LIN {X 0,Y 418.249,Z 282.699,A -85,B 0,C 180,E1 -10100.662,E2 -10100.662} C_VEL
LIN {X 0,Y 418.288,Z 282.694,A -85,B 0,C 180,E1 -10103.781,E2 -10103.781} C_VEL
LIN {X 0,Y 418.309,Z 282.695,A -85,B 0,C 180,E1 -10107.07,E2 -10107.07} C_VEL
LIN {X 0,Y 418.243,Z 282.698,A -85,B 0,C 180,E1 -10110.272,E2 -10110.272} C_VEL
LIN {X 0,Y 418.247,Z 282.697,A -85,B 0,C 180,E1 -10113.677,E2 -10113.677} C_VEL
LIN {X 0,Y 418.244,Z 282.692,A -85,B 0,C 180,E1 -10117.223,E2 -10117.223} C_VEL
LIN {X 0,Y 418.251,Z 282.695,A -85,B 0,C 180,E1 -10119.681,E2 -10119.681} C_VEL
LIN {X 0,Y 418.231,Z 282.701,A -85,B 0,C 180,E1 -10122.321,E2 -10122.321} C_VEL
LIN {X 0,Y 418.24,Z 282.698,A -85,B 0,C 180,E1 -10125.109,E2 -10125.109} C_VEL
LIN {X 0,Y 418.24,Z 282.695,A -85,B 0,C 180,E1 -10127.767,E2 -10127.767} C_VEL
LIN {X 0,Y 418.256,Z 282.699,A -85,B 0,C 180,E1 -10130.618,E2 -10130.618} C_VEL
LIN {X 0,Y 418.25,Z 282.714,A -85,B 0,C 180,E1 -10133.881,E2 -10133.881} C_VEL
LIN {X 0,Y 423.641,Z 299.97,A -85,B 0,C 180,E1 -10136.508,E2 -10136.508} C_VEL
LIN {X 0,Y 426.193,Z 308.268,A -85,B 0,C 180,E1 -10137.685,E2 -10137.685} C_VEL
LIN {X 0,Y 432.078,Z 321.178,A -85,B 0,C 180,E1 -10138.364,E2 -10138.364} C_VEL
LIN {X 0,Y 435.625,Z 342.848,A -85,B 0,C 180,E1 -10139.021,E2 -10139.021} C_VEL
LIN {X 0,Y 432.249,Z 513.22,A -85,B 0,C 180,E1 -10141.933,E2 -10141.933} C_VEL
LIN {X 0,Y 431.437,Z 530.001,A -85,B 0,C 180,E1 -10142.371,E2 -10142.371} C_VEL
LIN {X 0,Y 430.361,Z 546.409,A -85,B 0,C 180,E1 -10142.987,E2 -10142.987} C_VEL
LIN {X 0,Y 429.185,Z 561.958,A -85,B 0,C 180,E1 -10143.76,E2 -10143.76} C_VEL
LIN {X 0,Y 427.765,Z 577.137,A -85,B 0,C 180,E1 -10144.712,E2 -10144.712} C_VEL
LIN {X 0,Y 426.267,Z 591.185,A -85,B 0,C 180,E1 -10145.788,E2 -10145.788} C_VEL
LIN {X 0,Y 424.709,Z 605.609,A -85,B 0,C 180,E1 -10147.116,E2 -10147.116} C_VEL
LIN {X 0,Y 423.361,Z 617.281,A -85,B 0,C 180,E1 -10148.376,E2 -10148.376} C_VEL
LIN {X 0,Y 421.85,Z 630.208,A -85,B 0,C 180,E1 -10150.03,E2 -10150.03} C_VEL
LIN {X 0,Y 420.534,Z 641.484,A -85,B 0,C 180,E1 -10151.739,E2 -10151.739} C_VEL
LIN {X 0,Y 419.547,Z 651.141,A -85,B 0,C 180,E1 -10153.455,E2 -10153.455} C_VEL
LIN {X 0,Y 418.597,Z 660.507,A -85,B 0,C 180,E1 -10155.414,E2 -10155.414} C_VEL
LIN {X 0,Y 417.976,Z 668.29,A -85,B 0,C 180,E1 -10157.374,E2 -10157.374} C_VEL
LIN {X 0,Y 417.475,Z 674.7,A -85,B 0,C 180,E1 -10159.328,E2 -10159.328} C_VEL
LIN {X 0,Y 417.212,Z 679.955,A -85,B 0,C 180,E1 -10161.28,E2 -10161.28} C_VEL
LIN {X 0,Y 417.137,Z 684.944,A -85,B 0,C 180,E1 -10163.739,E2 -10163.739} C_VEL
LIN {X 0,Y 416.984,Z 688.178,A -85,B 0,C 180,E1 -10166.134,E2 -10166.134} C_VEL
LIN {X 0,Y 417.046,Z 689.646,A -85,B 0,C 180,E1 -10168.069,E2 -10168.069} C_VEL
LIN {X 0,Y 416.999,Z 690.206,A -85,B 0,C 180,E1 -10170,E2 -10170} C_VEL
LIN {X 0,Y 417.059,Z 689.728,A -85,B 0,C 180,E1 -10171.932,E2 -10171.932} C_VEL
LIN {X 0,Y 416.982,Z 688.348,A -85,B 0,C 180,E1 -10173.866,E2 -10173.866} C_VEL
LIN {X 0,Y 417.137,Z 685.222,A -85,B 0,C 180,E1 -10176.261,E2 -10176.261} C_VEL
LIN {X 0,Y 417.183,Z 681.492,A -85,B 0,C 180,E1 -10178.233,E2 -10178.233} C_VEL
LIN {X 0,Y 417.397,Z 676.77,A -85,B 0,C 180,E1 -10180.183,E2 -10180.183} C_VEL
LIN {X 0,Y 417.89,Z 670.825,A -85,B 0,C 180,E1 -10182.136,E2 -10182.136} C_VEL
LIN {X 0,Y 418.552,Z 662.671,A -85,B 0,C 180,E1 -10184.34,E2 -10184.34} C_VEL
LIN {X 0,Y 419.584,Z 653.944,A -85,B 0,C 180,E1 -10186.294,E2 -10186.294} C_VEL
LIN {X 0,Y 420.748,Z 643.558,A -85,B 0,C 180,E1 -10188.252,E2 -10188.252} C_VEL
LIN {X 0,Y 422.177,Z 632.774,A -85,B 0,C 180,E1 -10189.954,E2 -10189.954} C_VEL
LIN {X 0,Y 423.752,Z 620.449,A -85,B 0,C 180,E1 -10191.617,E2 -10191.617} C_VEL
LIN {X 0,Y 425.414,Z 607.474,A -85,B 0,C 180,E1 -10193.102,E2 -10193.102} C_VEL
LIN {X 0,Y 427.132,Z 593.835,A -85,B 0,C 180,E1 -10194.419,E2 -10194.419} C_VEL
LIN {X 0,Y 428.934,Z 578.449,A -85,B 0,C 180,E1 -10195.645,E2 -10195.645} C_VEL
LIN {X 0,Y 430.648,Z 562.514,A -85,B 0,C 180,E1 -10196.666,E2 -10196.666} C_VEL
LIN {X 0,Y 431.982,Z 547.62,A -85,B 0,C 180,E1 -10197.427,E2 -10197.427} C_VEL
LIN {X 0,Y 433.199,Z 531.35,A -85,B 0,C 180,E1 -10198.066,E2 -10198.066} C_VEL
LIN {X 0,Y 434.124,Z 514.455,A -85,B 0,C 180,E1 -10198.532,E2 -10198.532} C_VEL
LIN {X 0,Y 438.122,Z 343.991,A -85,B 0,C 180,E1 -10201.515,E2 -10201.515} C_VEL
LIN {X 0,Y 437.367,Z 337.587,A -85,B 0,C 180,E1 -10201.708,E2 -10201.708} C_VEL
LIN {X 0,Y 434.883,Z 323.612,A -85,B 0,C 180,E1 -10202.21,E2 -10202.21} C_VEL
LIN {X 0,Y 426.694,Z 307.126,A -85,B 0,C 180,E1 -10203.348,E2 -10203.348} C_VEL
LIN {X 0,Y 422.578,Z 294.815,A -85,B 0,C 180,E1 -10205.42,E2 -10205.42} C_VEL
LIN {X 0,Y 418.253,Z 282.699,A -85,B 0,C 180,E1 -10207.639,E2 -10207.639} C_VEL
LIN {X 0,Y 418.223,Z 282.701,A -85,B 0,C 180,E1 -10210.948,E2 -10210.948} C_VEL
LIN {X 0,Y 418.216,Z 282.702,A -85,B 0,C 180,E1 -10213.731,E2 -10213.731} C_VEL
LIN {X 0,Y 418.208,Z 282.702,A -85,B 0,C 180,E1 -10216.449,E2 -10216.449} C_VEL
LIN {X 0,Y 418.223,Z 282.692,A -85,B 0,C 180,E1 -10219.131,E2 -10219.131} C_VEL
LIN {X 0,Y 418.228,Z 282.69,A -85,B 0,C 180,E1 -10222.167,E2 -10222.167} C_VEL
LIN {X 0,Y 418.265,Z 282.693,A -85,B 0,C 180,E1 -10225.42,E2 -10225.42} C_VEL
LIN {X 0,Y 418.211,Z 282.699,A -85,B 0,C 180,E1 -10228.604,E2 -10228.604} C_VEL
LIN {X 0,Y 418.292,Z 282.672,A -85,B 0,C 180,E1 -10231.937,E2 -10231.937} C_VEL
LIN {X 0,Y 418.29,Z 282.69,A -85,B 0,C 180,E1 -10235.163,E2 -10235.163} C_VEL
LIN {X 0,Y 418.235,Z 282.685,A -85,B 0,C 180,E1 -10238.304,E2 -10238.304} C_VEL
LIN {X 0,Y 418.284,Z 282.687,A -85,B 0,C 180,E1 -10241.384,E2 -10241.384} C_VEL
LIN {X 0,Y 418.303,Z 282.677,A -85,B 0,C 180,E1 -10244.406,E2 -10244.406} C_VEL
LIN {X 0,Y 418.357,Z 282.679,A -85,B 0,C 180,E1 -10247.386,E2 -10247.386} C_VEL
LIN {X 0,Y 418.339,Z 282.668,A -85,B 0,C 180,E1 -10250.329,E2 -10250.329} C_VEL
LIN {X 0,Y 418.446,Z 282.67,A -85,B 0,C 180,E1 -10253.249,E2 -10253.249} C_VEL
LIN {X 0,Y 418.331,Z 282.664,A -85,B 0,C 180,E1 -10255.182,E2 -10255.182} C_VEL
LIN {X 0,Y 418.542,Z 282.658,A -85,B 0,C 180,E1 -10258.076,E2 -10258.076} C_VEL
LIN {X 0,Y 418.666,Z 282.644,A -85,B 0,C 180,E1 -10260.001,E2 -10260.001} C_VEL
LIN {X 0,Y 418.475,Z 282.654,A -85,B 0,C 180,E1 -10262.888,E2 -10262.888} C_VEL
LIN {X 0,Y 418.445,Z 282.663,A -85,B 0,C 180,E1 -10266.551,E2 -10266.551} C_VEL
LIN {X 0,Y 418.337,Z 282.679,A -85,B 0,C 180,E1 -10269.672,E2 -10269.672} C_VEL
LIN {X 0,Y 418.349,Z 282.671,A -85,B 0,C 180,E1 -10273.001,E2 -10273.001} C_VEL
LIN {X 0,Y 418.267,Z 282.696,A -85,B 0,C 180,E1 -10276.713,E2 -10276.713} C_VEL
LIN {X 0,Y 418.273,Z 282.679,A -85,B 0,C 180,E1 -10279.79,E2 -10279.79} C_VEL
LIN {X 0,Y 418.227,Z 282.694,A -85,B 0,C 180,E1 -10282.737,E2 -10282.737} C_VEL
LIN {X 0,Y 418.212,Z 282.703,A -85,B 0,C 180,E1 -10285.909,E2 -10285.909} C_VEL
LIN {X 0,Y 418.257,Z 282.692,A -85,B 0,C 180,E1 -10289.163,E2 -10289.163} C_VEL
LIN {X 0,Y 418.233,Z 282.693,A -85,B 0,C 180,E1 -10292.53,E2 -10292.53} C_VEL
LIN {X 0,Y 418.249,Z 282.695,A -85,B 0,C 180,E1 -10294.843,E2 -10294.843} C_VEL
LIN {X 0,Y 418.234,Z 282.695,A -85,B 0,C 180,E1 -10298.445,E2 -10298.445} C_VEL
LIN {X 0,Y 418.249,Z 282.867,A -85,B 0,C 180,E1 -10302.071,E2 -10302.071} C_VEL
LIN {X 0,Y 420.134,Z 288.122,A -85,B 0,C 180,E1 -10303.057,E2 -10303.057} C_VEL
LIN {X 0,Y 429.975,Z 305.451,A -85,B 0,C 180,E1 -10304.41,E2 -10304.41} C_VEL
LIN {X 0,Y 438.474,Z 322.374,A -85,B 0,C 180,E1 -10305.542,E2 -10305.542} C_VEL
LIN {X 0,Y 434.474,Z 493.566,A -85,B 0,C 180,E1 -10308.551,E2 -10308.551} C_VEL
LIN {X 0,Y 433.607,Z 510.226,A -85,B 0,C 180,E1 -10309.029,E2 -10309.029} C_VEL
LIN {X 0,Y 432.602,Z 524.979,A -85,B 0,C 180,E1 -10309.62,E2 -10309.62} C_VEL
LIN {X 0,Y 431.281,Z 540.752,A -85,B 0,C 180,E1 -10310.438,E2 -10310.438} C_VEL
LIN {X 0,Y 429.944,Z 554.135,A -85,B 0,C 180,E1 -10311.3,E2 -10311.3} C_VEL
LIN {X 0,Y 428.353,Z 568.136,A -85,B 0,C 180,E1 -10312.39,E2 -10312.39} C_VEL
LIN {X 0,Y 426.623,Z 582.554,A -85,B 0,C 180,E1 -10313.745,E2 -10313.745} C_VEL
LIN {X 0,Y 425.049,Z 594.567,A -85,B 0,C 180,E1 -10315.074,E2 -10315.074} C_VEL
LIN {X 0,Y 423.256,Z 607.49,A -85,B 0,C 180,E1 -10316.773,E2 -10316.773} C_VEL
LIN {X 0,Y 421.775,Z 618.26,A -85,B 0,C 180,E1 -10318.456,E2 -10318.456} C_VEL
LIN {X 0,Y 420.482,Z 628.576,A -85,B 0,C 180,E1 -10320.36,E2 -10320.36} C_VEL
LIN {X 0,Y 419.522,Z 636.327,A -85,B 0,C 180,E1 -10322.026,E2 -10322.026} C_VEL
LIN {X 0,Y 418.584,Z 644.425,A -85,B 0,C 180,E1 -10324.117,E2 -10324.117} C_VEL
LIN {X 0,Y 418.36,Z 646.637,A -85,B 0,C 180,E1 -10324.771,E2 -10324.771} C_VEL
LIN {X 0,Y 417.477,Z 649.095,A -85,B 0,C 180,E1 -10325.502,E2 -10325.502} C_VEL
LIN {X 0,Y 412.902,Z 654.191,A -85,B 0,C 180,E1 -10327.17,E2 -10327.17} C_VEL
LIN {X 0,Y 410.75,Z 656.686,A -85,B 0,C 180,E1 -10328.171,E2 -10328.171} C_VEL
LIN {X 0,Y 410.338,Z 657.819,A -85,B 0,C 180,E1 -10328.694,E2 -10328.694} C_VEL
LIN {X 0,Y 409.993,Z 661.815,A -85,B 0,C 180,E1 -10330.992,E2 -10330.992} C_VEL
LIN {X 0,Y 409.86,Z 664.298,A -85,B 0,C 180,E1 -10333.052,E2 -10333.052} C_VEL
LIN {X 0,Y 409.771,Z 665.655,A -85,B 0,C 180,E1 -10335.092,E2 -10335.092} C_VEL
LIN {X 0,Y 409.814,Z 666.051,A -85,B 0,C 180,E1 -10337.118,E2 -10337.118} C_VEL
LIN {X 0,Y 409.863,Z 665.421,A -85,B 0,C 180,E1 -10339.128,E2 -10339.128} C_VEL
LIN {X 0,Y 409.852,Z 663.842,A -85,B 0,C 180,E1 -10341.122,E2 -10341.122} C_VEL
LIN {X 0,Y 410.035,Z 661.259,A -85,B 0,C 180,E1 -10343.109,E2 -10343.109} C_VEL
LIN {X 0,Y 410.224,Z 657.666,A -85,B 0,C 180,E1 -10345.086,E2 -10345.086} C_VEL
LIN {X 0,Y 410.569,Z 653.047,A -85,B 0,C 180,E1 -10347.056,E2 -10347.056} C_VEL
LIN {X 0,Y 410.987,Z 647.259,A -85,B 0,C 180,E1 -10349.02,E2 -10349.02} C_VEL
LIN {X 0,Y 411.677,Z 640.303,A -85,B 0,C 180,E1 -10350.978,E2 -10350.978} C_VEL
LIN {X 0,Y 412.563,Z 631.963,A -85,B 0,C 180,E1 -10352.929,E2 -10352.929} C_VEL
LIN {X 0,Y 413.827,Z 622,A -85,B 0,C 180,E1 -10354.871,E2 -10354.871} C_VEL
LIN {X 0,Y 415.148,Z 611.773,A -85,B 0,C 180,E1 -10356.561,E2 -10356.561} C_VEL
LIN {X 0,Y 416.583,Z 599.856,A -85,B 0,C 180,E1 -10358.245,E2 -10358.245} C_VEL
LIN {X 0,Y 418.04,Z 587.883,A -85,B 0,C 180,E1 -10359.678,E2 -10359.678} C_VEL
LIN {X 0,Y 419.556,Z 574.948,A -85,B 0,C 180,E1 -10360.984,E2 -10360.984} C_VEL
LIN {X 0,Y 421.063,Z 561.104,A -85,B 0,C 180,E1 -10362.165,E2 -10362.165} C_VEL
LIN {X 0,Y 422.537,Z 546.137,A -85,B 0,C 180,E1 -10363.221,E2 -10363.221} C_VEL
LIN {X 0,Y 423.733,Z 530.732,A -85,B 0,C 180,E1 -10364.099,E2 -10364.099} C_VEL
LIN {X 0,Y 424.907,Z 514.713,A -85,B 0,C 180,E1 -10364.794,E2 -10364.794} C_VEL
LIN {X 0,Y 425.779,Z 498.352,A -85,B 0,C 180,E1 -10365.313,E2 -10365.313} C_VEL
LIN {X 0,Y 426.352,Z 478.659,A -85,B 0,C 180,E1 -10365.721,E2 -10365.721} C_VEL
LIN {X 0,Y 429.594,Z 323.165,A -85,B 0,C 180,E1 -10368.401,E2 -10368.401} C_VEL
LIN {X 0,Y 415.653,Z 293.917,A -85,B 0,C 180,E1 -10370.031,E2 -10370.031} C_VEL
LIN {X 0,Y 412.301,Z 287.377,A -85,B 0,C 180,E1 -10370.441,E2 -10370.441} C_VEL
LIN {X 0,Y 411.185,Z 283.575,A -85,B 0,C 180,E1 -10371.1,E2 -10371.1} C_VEL
LIN {X 0,Y 411.195,Z 283.582,A -85,B 0,C 180,E1 -10374.217,E2 -10374.217} C_VEL
LIN {X 0,Y 411.146,Z 283.584,A -85,B 0,C 180,E1 -10377.486,E2 -10377.486} C_VEL
LIN {X 0,Y 411.198,Z 283.576,A -85,B 0,C 180,E1 -10379.713,E2 -10379.713} C_VEL
LIN {X 0,Y 411.205,Z 283.575,A -85,B 0,C 180,E1 -10383.156,E2 -10383.156} C_VEL
LIN {X 0,Y 411.189,Z 283.578,A -85,B 0,C 180,E1 -10386.551,E2 -10386.551} C_VEL
LIN {X 0,Y 411.168,Z 283.58,A -85,B 0,C 180,E1 -10389.719,E2 -10389.719} C_VEL
LIN {X 0,Y 411.162,Z 283.576,A -85,B 0,C 180,E1 -10393.135,E2 -10393.135} C_VEL
LIN {X 0,Y 411.164,Z 283.574,A -85,B 0,C 180,E1 -10395.882,E2 -10395.882} C_VEL
LIN {X 0,Y 411.159,Z 283.582,A -85,B 0,C 180,E1 -10399.492,E2 -10399.492} C_VEL
LIN {X 0,Y 411.181,Z 283.551,A -85,B 0,C 180,E1 -10402.024,E2 -10402.024} C_VEL
LIN {X 0,Y 411.203,Z 283.555,A -85,B 0,C 180,E1 -10405.123,E2 -10405.123} C_VEL
LIN {X 0,Y 411.165,Z 283.583,A -85,B 0,C 180,E1 -10408.002,E2 -10408.002} C_VEL
LIN {X 0,Y 411.173,Z 283.569,A -85,B 0,C 180,E1 -10411.406,E2 -10411.406} C_VEL
LIN {X 0,Y 411.189,Z 283.573,A -85,B 0,C 180,E1 -10414.941,E2 -10414.941} C_VEL
LIN {X 0,Y 411.205,Z 283.575,A -85,B 0,C 180,E1 -10417.913,E2 -10417.913} C_VEL
LIN {X 0,Y 411.221,Z 283.569,A -85,B 0,C 180,E1 -10421.051,E2 -10421.051} C_VEL
LIN {X 0,Y 411.255,Z 283.568,A -85,B 0,C 180,E1 -10424.131,E2 -10424.131} C_VEL
LIN {X 0,Y 411.305,Z 283.559,A -85,B 0,C 180,E1 -10427.165,E2 -10427.165} C_VEL
LIN {X 0,Y 411.291,Z 283.563,A -85,B 0,C 180,E1 -10430.161,E2 -10430.161} C_VEL
LIN {X 0,Y 411.438,Z 283.543,A -85,B 0,C 180,E1 -10433.132,E2 -10433.132} C_VEL
LIN {X 0,Y 411.303,Z 283.552,A -85,B 0,C 180,E1 -10435.098,E2 -10435.098} C_VEL
LIN {X 0,Y 411.508,Z 283.535,A -85,B 0,C 180,E1 -10438.042,E2 -10438.042} C_VEL
LIN {X 0,Y 411.639,Z 283.507,A -85,B 0,C 180,E1 -10439.999,E2 -10439.999} C_VEL
LIN {X 0,Y 411.457,Z 283.543,A -85,B 0,C 180,E1 -10442.937,E2 -10442.937} C_VEL
LIN {X 0,Y 411.43,Z 283.531,A -85,B 0,C 180,E1 -10446.867,E2 -10446.867} C_VEL
LIN {X 0,Y 411.293,Z 283.564,A -85,B 0,C 180,E1 -10449.838,E2 -10449.838} C_VEL
LIN {X 0,Y 411.305,Z 283.562,A -85,B 0,C 180,E1 -10453.104,E2 -10453.104} C_VEL
LIN {X 0,Y 411.257,Z 283.569,A -85,B 0,C 180,E1 -10456.888,E2 -10456.888} C_VEL
LIN {X 0,Y 411.23,Z 283.572,A -85,B 0,C 180,E1 -10459.986,E2 -10459.986} C_VEL
LIN {X 0,Y 411.203,Z 283.579,A -85,B 0,C 180,E1 -10463.147,E2 -10463.147} C_VEL
LIN {X 0,Y 411.237,Z 283.571,A -85,B 0,C 180,E1 -10466.38,E2 -10466.38} C_VEL
LIN {X 0,Y 411.199,Z 283.576,A -85,B 0,C 180,E1 -10469.712,E2 -10469.712} C_VEL
LIN {X 0,Y 411.205,Z 283.576,A -85,B 0,C 180,E1 -10473.155,E2 -10473.155} C_VEL
LIN {X 0,Y 411.194,Z 283.568,A -85,B 0,C 180,E1 -10476.553,E2 -10476.553} C_VEL
LIN {X 0,Y 411.214,Z 283.571,A -85,B 0,C 180,E1 -10479.728,E2 -10479.728} C_VEL
LIN {X 0,Y 411.176,Z 283.58,A -85,B 0,C 180,E1 -10483.133,E2 -10483.133} C_VEL
LIN {X 0,Y 411.172,Z 283.581,A -85,B 0,C 180,E1 -10485.88,E2 -10485.88} C_VEL
LIN {X 0,Y 411.164,Z 283.584,A -85,B 0,C 180,E1 -10488.771,E2 -10488.771} C_VEL
LIN {X 0,Y 411.205,Z 283.574,A -85,B 0,C 180,E1 -10491.831,E2 -10491.831} C_VEL
LIN {X 0,Y 411.195,Z 283.636,A -85,B 0,C 180,E1 -10493.395,E2 -10493.395} C_VEL
LIN {X 0,Y 416.856,Z 301.621,A -85,B 0,C 180,E1 -10496.195,E2 -10496.195} C_VEL
LIN {X 0,Y 418.756,Z 307.842,A -85,B 0,C 180,E1 -10497.108,E2 -10497.108} C_VEL
LIN {X 0,Y 426.119,Z 323.923,A -85,B 0,C 180,E1 -10497.978,E2 -10497.978} C_VEL
LIN {X 0,Y 429.371,Z 343.747,A -85,B 0,C 180,E1 -10498.591,E2 -10498.591} C_VEL
LIN {X 0,Y 425.808,Z 513.76,A -85,B 0,C 180,E1 -10501.538,E2 -10501.538} C_VEL
LIN {X 0,Y 424.982,Z 530.254,A -85,B 0,C 180,E1 -10501.981,E2 -10501.981} C_VEL
LIN {X 0,Y 423.857,Z 546.546,A -85,B 0,C 180,E1 -10502.605,E2 -10502.605} C_VEL
LIN {X 0,Y 422.631,Z 562.034,A -85,B 0,C 180,E1 -10503.388,E2 -10503.388} C_VEL
LIN {X 0,Y 421.112,Z 577.643,A -85,B 0,C 180,E1 -10504.383,E2 -10504.383} C_VEL
LIN {X 0,Y 419.535,Z 591.941,A -85,B 0,C 180,E1 -10505.505,E2 -10505.505} C_VEL
LIN {X 0,Y 417.919,Z 606.203,A -85,B 0,C 180,E1 -10506.853,E2 -10506.853} C_VEL
LIN {X 0,Y 416.433,Z 618.342,A -85,B 0,C 180,E1 -10508.205,E2 -10508.205} C_VEL
LIN {X 0,Y 415.047,Z 629.704,A -85,B 0,C 180,E1 -10509.688,E2 -10509.688} C_VEL
LIN {X 0,Y 413.66,Z 641.03,A -85,B 0,C 180,E1 -10511.424,E2 -10511.424} C_VEL
LIN {X 0,Y 412.482,Z 651.988,A -85,B 0,C 180,E1 -10513.418,E2 -10513.418} C_VEL
LIN {X 0,Y 411.496,Z 661.173,A -85,B 0,C 180,E1 -10515.409,E2 -10515.409} C_VEL
LIN {X 0,Y 410.966,Z 667.957,A -85,B 0,C 180,E1 -10517.155,E2 -10517.155} C_VEL
LIN {X 0,Y 410.424,Z 674.397,A -85,B 0,C 180,E1 -10519.143,E2 -10519.143} C_VEL
LIN {X 0,Y 410.146,Z 679.676,A -85,B 0,C 180,E1 -10521.129,E2 -10521.129} C_VEL
LIN {X 0,Y 410.041,Z 683.737,A -85,B 0,C 180,E1 -10523.109,E2 -10523.109} C_VEL
LIN {X 0,Y 409.951,Z 686.799,A -85,B 0,C 180,E1 -10525.083,E2 -10525.083} C_VEL
LIN {X 0,Y 409.908,Z 688.788,A -85,B 0,C 180,E1 -10527.052,E2 -10527.052} C_VEL
LIN {X 0,Y 409.93,Z 689.838,A -85,B 0,C 180,E1 -10529.018,E2 -10529.018} C_VEL
LIN {X 0,Y 409.933,Z 689.872,A -85,B 0,C 180,E1 -10530.982,E2 -10530.982} C_VEL
LIN {X 0,Y 409.904,Z 688.982,A -85,B 0,C 180,E1 -10532.949,E2 -10532.949} C_VEL
LIN {X 0,Y 409.934,Z 687.072,A -85,B 0,C 180,E1 -10534.918,E2 -10534.918} C_VEL
LIN {X 0,Y 410.04,Z 684.209,A -85,B 0,C 180,E1 -10536.891,E2 -10536.891} C_VEL
LIN {X 0,Y 410.152,Z 680.271,A -85,B 0,C 180,E1 -10538.871,E2 -10538.871} C_VEL
LIN {X 0,Y 410.458,Z 675.262,A -85,B 0,C 180,E1 -10540.856,E2 -10540.856} C_VEL
LIN {X 0,Y 411.038,Z 668.776,A -85,B 0,C 180,E1 -10542.945,E2 -10542.945} C_VEL
LIN {X 0,Y 411.93,Z 659.569,A -85,B 0,C 180,E1 -10545.334,E2 -10545.334} C_VEL
LIN {X 0,Y 413.034,Z 650.495,A -85,B 0,C 180,E1 -10547.267,E2 -10547.267} C_VEL
LIN {X 0,Y 414.283,Z 640.617,A -85,B 0,C 180,E1 -10549.06,E2 -10549.06} C_VEL
LIN {X 0,Y 415.845,Z 629.479,A -85,B 0,C 180,E1 -10550.788,E2 -10550.788} C_VEL
LIN {X 0,Y 417.419,Z 618.165,A -85,B 0,C 180,E1 -10552.285,E2 -10552.285} C_VEL
LIN {X 0,Y 419.176,Z 605.348,A -85,B 0,C 180,E1 -10553.728,E2 -10553.728} C_VEL
LIN {X 0,Y 420.857,Z 592.715,A -85,B 0,C 180,E1 -10554.939,E2 -10554.939} C_VEL
LIN {X 0,Y 422.722,Z 577.804,A -85,B 0,C 180,E1 -10556.133,E2 -10556.133} C_VEL
LIN {X 0,Y 424.34,Z 563.011,A -85,B 0,C 180,E1 -10557.095,E2 -10557.095} C_VEL
LIN {X 0,Y 425.73,Z 548.365,A -85,B 0,C 180,E1 -10557.865,E2 -10557.865} C_VEL
LIN {X 0,Y 427.067,Z 531.646,A -85,B 0,C 180,E1 -10558.538,E2 -10558.538} C_VEL
LIN {X 0,Y 428.048,Z 514.763,A -85,B 0,C 180,E1 -10559.016,E2 -10559.016} C_VEL
LIN {X 0,Y 430.047,Z 433.281,A -85,B 0,C 180,E1 -10560.472,E2 -10560.472} C_VEL
LIN {X 0,Y 432.184,Z 343.222,A -85,B 0,C 180,E1 -10562.067,E2 -10562.067} C_VEL
LIN {X 0,Y 429.461,Z 326.894,A -85,B 0,C 180,E1 -10562.653,E2 -10562.653} C_VEL
LIN {X 0,Y 421.555,Z 311.061,A -85,B 0,C 180,E1 -10563.759,E2 -10563.759} C_VEL
LIN {X 0,Y 419.451,Z 306.924,A -85,B 0,C 180,E1 -10564.078,E2 -10564.078} C_VEL
LIN {X 0,Y 414.987,Z 293.984,A -85,B 0,C 180,E1 -10566.352,E2 -10566.352} C_VEL
LIN {X 0,Y 411.217,Z 283.575,A -85,B 0,C 180,E1 -10568.332,E2 -10568.332} C_VEL
LIN {X 0,Y 411.178,Z 283.57,A -85,B 0,C 180,E1 -10571.806,E2 -10571.806} C_VEL
LIN {X 0,Y 411.176,Z 283.57,A -85,B 0,C 180,E1 -10575.51,E2 -10575.51} C_VEL
LIN {X 0,Y 411.163,Z 283.569,A -85,B 0,C 180,E1 -10578.772,E2 -10578.772} C_VEL
LIN {X 0,Y 411.206,Z 283.567,A -85,B 0,C 180,E1 -10581.832,E2 -10581.832} C_VEL
LIN {X 0,Y 411.211,Z 283.574,A -85,B 0,C 180,E1 -10585.122,E2 -10585.122} C_VEL
LIN {X 0,Y 411.165,Z 283.572,A -85,B 0,C 180,E1 -10588.003,E2 -10588.003} C_VEL
LIN {X 0,Y 411.218,Z 283.555,A -85,B 0,C 180,E1 -10591.411,E2 -10591.411} C_VEL
LIN {X 0,Y 411.239,Z 283.569,A -85,B 0,C 180,E1 -10593.62,E2 -10593.62} C_VEL
LIN {X 0,Y 411.198,Z 283.557,A -85,B 0,C 180,E1 -10596.853,E2 -10596.853} C_VEL
LIN {X 0,Y 411.216,Z 283.573,A -85,B 0,C 180,E1 -10600.051,E2 -10600.051} C_VEL
LIN {X 0,Y 411.264,Z 283.546,A -85,B 0,C 180,E1 -10603.132,E2 -10603.132} C_VEL
LIN {X 0,Y 411.307,Z 283.561,A -85,B 0,C 180,E1 -10606.896,E2 -10606.896} C_VEL
LIN {X 0,Y 411.292,Z 283.544,A -85,B 0,C 180,E1 -10610.162,E2 -10610.162} C_VEL
LIN {X 0,Y 411.395,Z 283.549,A -85,B 0,C 180,E1 -10613.132,E2 -10613.132} C_VEL
LIN {X 0,Y 411.302,Z 283.54,A -85,B 0,C 180,E1 -10615.099,E2 -10615.099} C_VEL
LIN {X 0,Y 411.511,Z 283.534,A -85,B 0,C 180,E1 -10618.043,E2 -10618.043} C_VEL
LIN {X 0,Y 411.636,Z 283.519,A -85,B 0,C 180,E1 -10620.001,E2 -10620.001} C_VEL
LIN {X 0,Y 411.433,Z 283.531,A -85,B 0,C 180,E1 -10622.938,E2 -10622.938} C_VEL
LIN {X 0,Y 411.394,Z 283.542,A -85,B 0,C 180,E1 -10626.549,E2 -10626.549} C_VEL
LIN {X 0,Y 411.319,Z 283.545,A -85,B 0,C 180,E1 -10628.847,E2 -10628.847} C_VEL
LIN {X 0,Y 411.285,Z 283.567,A -85,B 0,C 180,E1 -10631.833,E2 -10631.833} C_VEL
LIN {X 0,Y 411.243,Z 283.559,A -85,B 0,C 180,E1 -10634.854,E2 -10634.854} C_VEL
LIN {X 0,Y 411.217,Z 283.565,A -85,B 0,C 180,E1 -10637.917,E2 -10637.917} C_VEL
LIN {X 0,Y 411.198,Z 283.575,A -85,B 0,C 180,E1 -10641.035,E2 -10641.035} C_VEL
LIN {X 0,Y 411.176,Z 283.565,A -85,B 0,C 180,E1 -10644.219,E2 -10644.219} C_VEL
LIN {X 0,Y 411.143,Z 283.576,A -85,B 0,C 180,E1 -10647.487,E2 -10647.487} C_VEL
LIN {X 0,Y 411.195,Z 283.575,A -85,B 0,C 180,E1 -10649.714,E2 -10649.714} C_VEL
LIN {X 0,Y 411.205,Z 283.575,A -85,B 0,C 180,E1 -10653.157,E2 -10653.157} C_VEL
LIN {X 0,Y 411.189,Z 283.579,A -85,B 0,C 180,E1 -10656.552,E2 -10656.552} C_VEL
LIN {X 0,Y 411.169,Z 283.584,A -85,B 0,C 180,E1 -10659.72,E2 -10659.72} C_VEL
LIN {X 0,Y 411.171,Z 283.679,A -85,B 0,C 180,E1 -10661.368,E2 -10661.368} C_VEL
LIN {X 0,Y 412.853,Z 288.495,A -85,B 0,C 180,E1 -10662.281,E2 -10662.281} C_VEL
LIN {X 0,Y 421,Z 302.29,A -85,B 0,C 180,E1 -10663.448,E2 -10663.448} C_VEL
LIN {X 0,Y 429.588,Z 318.34,A -85,B 0,C 180,E1 -10664.635,E2 -10664.635} C_VEL
LIN {X 0,Y 432.6,Z 324.72,A -85,B 0,C 180,E1 -10665.05,E2 -10665.05} C_VEL
LIN {X 0,Y 428.447,Z 493.526,A -85,B 0,C 180,E1 -10668.053,E2 -10668.053} C_VEL
LIN {X 0,Y 427.519,Z 510.221,A -85,B 0,C 180,E1 -10668.533,E2 -10668.533} C_VEL
LIN {X 0,Y 426.551,Z 524.023,A -85,B 0,C 180,E1 -10669.085,E2 -10669.085} C_VEL
LIN {X 0,Y 425.241,Z 539.319,A -85,B 0,C 180,E1 -10669.867,E2 -10669.867} C_VEL
LIN {X 0,Y 423.737,Z 553.456,A -85,B 0,C 180,E1 -10670.777,E2 -10670.777} C_VEL
LIN {X 0,Y 421.994,Z 568.502,A -85,B 0,C 180,E1 -10671.96,E2 -10671.96} C_VEL
LIN {X 0,Y 420.202,Z 582.575,A -85,B 0,C 180,E1 -10673.298,E2 -10673.298} C_VEL
LIN {X 0,Y 418.437,Z 595.327,A -85,B 0,C 180,E1 -10674.735,E2 -10674.735} C_VEL
LIN {X 0,Y 416.556,Z 608.179,A -85,B 0,C 180,E1 -10676.458,E2 -10676.458} C_VEL
LIN {X 0,Y 414.903,Z 619.783,A -85,B 0,C 180,E1 -10678.324,E2 -10678.324} C_VEL
LIN {X 0,Y 413.644,Z 628.893,A -85,B 0,C 180,E1 -10680.057,E2 -10680.057} C_VEL
LIN {X 0,Y 412.456,Z 637.789,A -85,B 0,C 180,E1 -10682.039,E2 -10682.039} C_VEL
LIN {X 0,Y 411.527,Z 645.775,A -85,B 0,C 180,E1 -10684.184,E2 -10684.184} C_VEL
LIN {X 0,Y 410.813,Z 652.146,A -85,B 0,C 180,E1 -10686.295,E2 -10686.295} C_VEL
LIN {X 0,Y 410.399,Z 657.189,A -85,B 0,C 180,E1 -10688.396,E2 -10688.396} C_VEL
LIN {X 0,Y 410.338,Z 657.819,A -85,B 0,C 180,E1 -10688.694,E2 -10688.694} C_VEL
LIN {X 0,Y 409.541,Z 659.442,A -85,B 0,C 180,E1 -10689.479,E2 -10689.479} C_VEL
LIN {X 0,Y 406.508,Z 661.801,A -85,B 0,C 180,E1 -10690.762,E2 -10690.762} C_VEL
LIN {X 0,Y 403.982,Z 663.319,A -85,B 0,C 180,E1 -10691.809,E2 -10691.809} C_VEL
LIN {X 0,Y 402.875,Z 664.211,A -85,B 0,C 180,E1 -10692.627,E2 -10692.627} C_VEL
LIN {X 0,Y 402.771,Z 664.453,A -85,B 0,C 180,E1 -10692.906,E2 -10692.906} C_VEL
LIN {X 0,Y 402.698,Z 665.772,A -85,B 0,C 180,E1 -10694.824,E2 -10694.824} C_VEL
LIN {X 0,Y 402.707,Z 666.289,A -85,B 0,C 180,E1 -10696.887,E2 -10696.887} C_VEL
LIN {X 0,Y 402.767,Z 665.721,A -85,B 0,C 180,E1 -10698.934,E2 -10698.934} C_VEL
LIN {X 0,Y 402.758,Z 664.262,A -85,B 0,C 180,E1 -10700.964,E2 -10700.964} C_VEL
LIN {X 0,Y 402.945,Z 661.739,A -85,B 0,C 180,E1 -10702.987,E2 -10702.987} C_VEL
LIN {X 0,Y 403.142,Z 658.268,A -85,B 0,C 180,E1 -10704.999,E2 -10704.999} C_VEL
LIN {X 0,Y 403.477,Z 653.714,A -85,B 0,C 180,E1 -10707.004,E2 -10707.004} C_VEL
LIN {X 0,Y 403.898,Z 648.062,A -85,B 0,C 180,E1 -10709.003,E2 -10709.003} C_VEL
LIN {X 0,Y 404.621,Z 641.244,A -85,B 0,C 180,E1 -10710.995,E2 -10710.995} C_VEL
LIN {X 0,Y 405.665,Z 631.896,A -85,B 0,C 180,E1 -10713.228,E2 -10713.228} C_VEL
LIN {X 0,Y 407.011,Z 621.869,A -85,B 0,C 180,E1 -10715.201,E2 -10715.201} C_VEL
LIN {X 0,Y 408.386,Z 611.564,A -85,B 0,C 180,E1 -10716.919,E2 -10716.919} C_VEL
LIN {X 0,Y 409.903,Z 599.546,A -85,B 0,C 180,E1 -10718.628,E2 -10718.628} C_VEL
LIN {X 0,Y 411.586,Z 586.384,A -85,B 0,C 180,E1 -10720.204,E2 -10720.204} C_VEL
LIN {X 0,Y 413.288,Z 571.929,A -85,B 0,C 180,E1 -10721.65,E2 -10721.65} C_VEL
LIN {X 0,Y 414.972,Z 557.35,A -85,B 0,C 180,E1 -10722.843,E2 -10722.843} C_VEL
LIN {X 0,Y 416.264,Z 543.349,A -85,B 0,C 180,E1 -10723.797,E2 -10723.797} C_VEL
LIN {X 0,Y 417.512,Z 528.366,A -85,B 0,C 180,E1 -10724.625,E2 -10724.625} C_VEL
LIN {X 0,Y 418.63,Z 512.532,A -85,B 0,C 180,E1 -10725.301,E2 -10725.301} C_VEL
LIN {X 0,Y 419.517,Z 496.076,A -85,B 0,C 180,E1 -10725.797,E2 -10725.797} C_VEL
LIN {X 0,Y 420.16,Z 471.614,A -85,B 0,C 180,E1 -10726.271,E2 -10726.271} C_VEL
LIN {X 0,Y 423.265,Z 325.078,A -85,B 0,C 180,E1 -10728.835,E2 -10728.835} C_VEL
LIN {X 0,Y 410.208,Z 297.646,A -85,B 0,C 180,E1 -10730.397,E2 -10730.397} C_VEL
LIN {X 0,Y 405.072,Z 287.407,A -85,B 0,C 180,E1 -10731.065,E2 -10731.065} C_VEL
LIN {X 0,Y 404.156,Z 284.444,A -85,B 0,C 180,E1 -10731.619,E2 -10731.619} C_VEL
LIN {X 0,Y 404.139,Z 284.455,A -85,B 0,C 180,E1 -10734.668,E2 -10734.668} C_VEL
LIN {X 0,Y 404.104,Z 284.466,A -85,B 0,C 180,E1 -10738.006,E2 -10738.006} C_VEL
LIN {X 0,Y 404.144,Z 284.46,A -85,B 0,C 180,E1 -10740.285,E2 -10740.285} C_VEL
LIN {X 0,Y 404.138,Z 284.46,A -85,B 0,C 180,E1 -10743.813,E2 -10743.813} C_VEL
LIN {X 0,Y 404.131,Z 284.455,A -85,B 0,C 180,E1 -10746.873,E2 -10746.873} C_VEL
LIN {X 0,Y 404.119,Z 284.461,A -85,B 0,C 180,E1 -10750.074,E2 -10750.074} C_VEL
LIN {X 0,Y 404.142,Z 284.45,A -85,B 0,C 180,E1 -10753.081,E2 -10753.081} C_VEL
LIN {X 0,Y 404.121,Z 284.451,A -85,B 0,C 180,E1 -10755.921,E2 -10755.921} C_VEL
LIN {X 0,Y 404.102,Z 284.459,A -85,B 0,C 180,E1 -10758.632,E2 -10758.632} C_VEL
LIN {X 0,Y 404.138,Z 284.436,A -85,B 0,C 180,E1 -10761.495,E2 -10761.495} C_VEL
LIN {X 0,Y 404.174,Z 284.429,A -85,B 0,C 180,E1 -10764.982,E2 -10764.982} C_VEL
LIN {X 0,Y 404.139,Z 284.454,A -85,B 0,C 180,E1 -10768.442,E2 -10768.442} C_VEL
LIN {X 0,Y 404.15,Z 284.441,A -85,B 0,C 180,E1 -10770.862,E2 -10770.862} C_VEL
LIN {X 0,Y 404.155,Z 284.449,A -85,B 0,C 180,E1 -10774.722,E2 -10774.722} C_VEL
LIN {X 0,Y 404.168,Z 284.445,A -85,B 0,C 180,E1 -10777.507,E2 -10777.507} C_VEL
LIN {X 0,Y 404.164,Z 284.447,A -85,B 0,C 180,E1 -10780.707,E2 -10780.707} C_VEL
LIN {X 0,Y 404.222,Z 284.445,A -85,B 0,C 180,E1 -10783.848,E2 -10783.848} C_VEL
LIN {X 0,Y 404.284,Z 284.433,A -85,B 0,C 180,E1 -10786.938,E2 -10786.938} C_VEL
LIN {X 0,Y 404.257,Z 284.44,A -85,B 0,C 180,E1 -10789.988,E2 -10789.988} C_VEL
LIN {X 0,Y 404.388,Z 284.422,A -85,B 0,C 180,E1 -10793.012,E2 -10793.012} C_VEL
LIN {X 0,Y 404.276,Z 284.426,A -85,B 0,C 180,E1 -10795.013,E2 -10795.013} C_VEL
LIN {X 0,Y 404.477,Z 284.411,A -85,B 0,C 180,E1 -10798.008,E2 -10798.008} C_VEL
LIN {X 0,Y 404.608,Z 284.382,A -85,B 0,C 180,E1 -10799.999,E2 -10799.999} C_VEL
LIN {X 0,Y 404.415,Z 284.42,A -85,B 0,C 180,E1 -10802.988,E2 -10802.988} C_VEL
LIN {X 0,Y 404.38,Z 284.408,A -85,B 0,C 180,E1 -10806.987,E2 -10806.987} C_VEL
LIN {X 0,Y 404.258,Z 284.439,A -85,B 0,C 180,E1 -10810.011,E2 -10810.011} C_VEL
LIN {X 0,Y 404.266,Z 284.44,A -85,B 0,C 180,E1 -10813.211,E2 -10813.211} C_VEL
LIN {X 0,Y 404.215,Z 284.447,A -85,B 0,C 180,E1 -10817.006,E2 -10817.006} C_VEL
LIN {X 0,Y 404.163,Z 284.452,A -85,B 0,C 180,E1 -10820.351,E2 -10820.351} C_VEL
LIN {X 0,Y 404.169,Z 284.454,A -85,B 0,C 180,E1 -10823.574,E2 -10823.574} C_VEL
LIN {X 0,Y 404.183,Z 284.451,A -85,B 0,C 180,E1 -10825.766,E2 -10825.766} C_VEL
LIN {X 0,Y 404.194,Z 284.445,A -85,B 0,C 180,E1 -10827.999,E2 -10827.999} C_VEL
LIN {X 0,Y 404.138,Z 284.457,A -85,B 0,C 180,E1 -10831.558,E2 -10831.558} C_VEL
LIN {X 0,Y 404.184,Z 284.45,A -85,B 0,C 180,E1 -10835.016,E2 -10835.016} C_VEL
LIN {X 0,Y 404.156,Z 284.456,A -85,B 0,C 180,E1 -10838.756,E2 -10838.756} C_VEL
LIN {X 0,Y 404.123,Z 284.456,A -85,B 0,C 180,E1 -10841.6,E2 -10841.6} C_VEL
LIN {X 0,Y 404.149,Z 284.449,A -85,B 0,C 180,E1 -10844.523,E2 -10844.523} C_VEL
LIN {X 0,Y 404.138,Z 284.451,A -85,B 0,C 180,E1 -10847.296,E2 -10847.296} C_VEL
LIN {X 0,Y 404.167,Z 284.453,A -85,B 0,C 180,E1 -10849.955,E2 -10849.955} C_VEL
LIN {X 0,Y 404.151,Z 284.625,A -85,B 0,C 180,E1 -10852.904,E2 -10852.904} C_VEL
LIN {X 0,Y 409.98,Z 302.784,A -85,B 0,C 180,E1 -10855.803,E2 -10855.803} C_VEL
LIN {X 0,Y 411.414,Z 307.69,A -85,B 0,C 180,E1 -10856.521,E2 -10856.521} C_VEL
LIN {X 0,Y 420.053,Z 326.307,A -85,B 0,C 180,E1 -10857.566,E2 -10857.566} C_VEL
LIN {X 0,Y 423.135,Z 344.937,A -85,B 0,C 180,E1 -10858.156,E2 -10858.156} C_VEL
LIN {X 0,Y 419.402,Z 514.305,A -85,B 0,C 180,E1 -10861.131,E2 -10861.131} C_VEL
LIN {X 0,Y 418.549,Z 530.506,A -85,B 0,C 180,E1 -10861.58,E2 -10861.58} C_VEL
LIN {X 0,Y 417.373,Z 546.663,A -85,B 0,C 180,E1 -10862.211,E2 -10862.211} C_VEL
LIN {X 0,Y 416.099,Z 562.074,A -85,B 0,C 180,E1 -10863.004,E2 -10863.004} C_VEL
LIN {X 0,Y 414.469,Z 578.152,A -85,B 0,C 180,E1 -10864.049,E2 -10864.049} C_VEL
LIN {X 0,Y 412.795,Z 592.634,A -85,B 0,C 180,E1 -10865.213,E2 -10865.213} C_VEL
LIN {X 0,Y 411.138,Z 606.749,A -85,B 0,C 180,E1 -10866.582,E2 -10866.582} C_VEL
LIN {X 0,Y 409.48,Z 619.547,A -85,B 0,C 180,E1 -10868.051,E2 -10868.051} C_VEL
LIN {X 0,Y 408.052,Z 630.978,A -85,B 0,C 180,E1 -10869.588,E2 -10869.588} C_VEL
LIN {X 0,Y 406.633,Z 642.086,A -85,B 0,C 180,E1 -10871.353,E2 -10871.353} C_VEL
LIN {X 0,Y 405.546,Z 651.576,A -85,B 0,C 180,E1 -10873.126,E2 -10873.126} C_VEL
LIN {X 0,Y 404.511,Z 660.799,A -85,B 0,C 180,E1 -10875.151,E2 -10875.151} C_VEL
LIN {X 0,Y 403.896,Z 667.912,A -85,B 0,C 180,E1 -10877.013,E2 -10877.013} C_VEL
LIN {X 0,Y 403.385,Z 674.077,A -85,B 0,C 180,E1 -10878.951,E2 -10878.951} C_VEL
LIN {X 0,Y 403.051,Z 679.385,A -85,B 0,C 180,E1 -10880.971,E2 -10880.971} C_VEL
LIN {X 0,Y 402.961,Z 683.467,A -85,B 0,C 180,E1 -10882.988,E2 -10882.988} C_VEL
LIN {X 0,Y 402.865,Z 686.553,A -85,B 0,C 180,E1 -10884.996,E2 -10884.996} C_VEL
LIN {X 0,Y 402.807,Z 688.554,A -85,B 0,C 180,E1 -10887,E2 -10887} C_VEL
LIN {X 0,Y 402.857,Z 689.626,A -85,B 0,C 180,E1 -10889.001,E2 -10889.001} C_VEL
LIN {X 0,Y 402.86,Z 689.669,A -85,B 0,C 180,E1 -10891,E2 -10891} C_VEL
LIN {X 0,Y 402.803,Z 688.8,A -85,B 0,C 180,E1 -10893.001,E2 -10893.001} C_VEL
LIN {X 0,Y 402.851,Z 686.902,A -85,B 0,C 180,E1 -10895.004,E2 -10895.004} C_VEL
LIN {X 0,Y 402.96,Z 684.065,A -85,B 0,C 180,E1 -10897.013,E2 -10897.013} C_VEL
LIN {X 0,Y 403.064,Z 680.143,A -85,B 0,C 180,E1 -10899.029,E2 -10899.029} C_VEL
LIN {X 0,Y 403.415,Z 675.161,A -85,B 0,C 180,E1 -10901.048,E2 -10901.048} C_VEL
LIN {X 0,Y 403.99,Z 669.02,A -85,B 0,C 180,E1 -10903.071,E2 -10903.071} C_VEL
LIN {X 0,Y 404.873,Z 660.536,A -85,B 0,C 180,E1 -10905.35,E2 -10905.35} C_VEL
LIN {X 0,Y 406.024,Z 651.605,A -85,B 0,C 180,E1 -10907.34,E2 -10907.34} C_VEL
LIN {X 0,Y 407.285,Z 642.156,A -85,B 0,C 180,E1 -10909.139,E2 -10909.139} C_VEL
LIN {X 0,Y 408.922,Z 631.284,A -85,B 0,C 180,E1 -10910.893,E2 -10910.893} C_VEL
LIN {X 0,Y 410.74,Z 618.652,A -85,B 0,C 180,E1 -10912.62,E2 -10912.62} C_VEL
LIN {X 0,Y 412.663,Z 605.558,A -85,B 0,C 180,E1 -10914.126,E2 -10914.126} C_VEL
LIN {X 0,Y 414.225,Z 594.403,A -85,B 0,C 180,E1 -10915.232,E2 -10915.232} C_VEL
LIN {X 0,Y 416.056,Z 580.216,A -85,B 0,C 180,E1 -10916.413,E2 -10916.413} C_VEL
LIN {X 0,Y 417.835,Z 565.567,A -85,B 0,C 180,E1 -10917.416,E2 -10917.416} C_VEL
LIN {X 0,Y 419.405,Z 550.484,A -85,B 0,C 180,E1 -10918.255,E2 -10918.255} C_VEL
LIN {X 0,Y 420.828,Z 533.743,A -85,B 0,C 180,E1 -10918.968,E2 -10918.968} C_VEL
LIN {X 0,Y 421.956,Z 516.233,A -85,B 0,C 180,E1 -10919.485,E2 -10919.485} C_VEL
LIN {X 0,Y 422.884,Z 484.65,A -85,B 0,C 180,E1 -10920.078,E2 -10920.078} C_VEL
LIN {X 0,Y 426.409,Z 344.695,A -85,B 0,C 180,E1 -10922.582,E2 -10922.582} C_VEL
LIN {X 0,Y 424.006,Z 329.943,A -85,B 0,C 180,E1 -10923.119,E2 -10923.119} C_VEL
LIN {X 0,Y 416.422,Z 314.805,A -85,B 0,C 180,E1 -10924.211,E2 -10924.211} C_VEL
LIN {X 0,Y 412.17,Z 306.761,A -85,B 0,C 180,E1 -10924.844,E2 -10924.844} C_VEL
LIN {X 0,Y 407.159,Z 292.615,A -85,B 0,C 180,E1 -10927.439,E2 -10927.439} C_VEL
LIN {X 0,Y 404.202,Z 284.442,A -85,B 0,C 180,E1 -10929.072,E2 -10929.072} C_VEL
LIN {X 0,Y 404.156,Z 284.452,A -85,B 0,C 180,E1 -10933.085,E2 -10933.085} C_VEL
LIN {X 0,Y 404.148,Z 284.449,A -85,B 0,C 180,E1 -10935.927,E2 -10935.927} C_VEL
LIN {X 0,Y 404.118,Z 284.446,A -85,B 0,C 180,E1 -10938.635,E2 -10938.635} C_VEL
LIN {X 0,Y 404.154,Z 284.448,A -85,B 0,C 180,E1 -10941.492,E2 -10941.492} C_VEL
LIN {X 0,Y 404.184,Z 284.451,A -85,B 0,C 180,E1 -10944.984,E2 -10944.984} C_VEL
LIN {X 0,Y 404.142,Z 284.45,A -85,B 0,C 180,E1 -10948.554,E2 -10948.554} C_VEL
LIN {X 0,Y 404.195,Z 284.427,A -85,B 0,C 180,E1 -10952.001,E2 -10952.001} C_VEL
LIN {X 0,Y 404.175,Z 284.447,A -85,B 0,C 180,E1 -10955.335,E2 -10955.335} C_VEL
LIN {X 0,Y 404.139,Z 284.442,A -85,B 0,C 180,E1 -10958.581,E2 -10958.581} C_VEL
LIN {X 0,Y 404.211,Z 284.44,A -85,B 0,C 180,E1 -10961.763,E2 -10961.763} C_VEL
LIN {X 0,Y 404.207,Z 284.439,A -85,B 0,C 180,E1 -10964.883,E2 -10964.883} C_VEL
LIN {X 0,Y 404.257,Z 284.43,A -85,B 0,C 180,E1 -10967.959,E2 -10967.959} C_VEL
LIN {X 0,Y 404.267,Z 284.431,A -85,B 0,C 180,E1 -10970.999,E2 -10970.999} C_VEL
LIN {X 0,Y 404.383,Z 284.417,A -85,B 0,C 180,E1 -10974.015,E2 -10974.015} C_VEL
LIN {X 0,Y 404.48,Z 284.409,A -85,B 0,C 180,E1 -10978.009,E2 -10978.009} C_VEL
LIN {X 0,Y 404.605,Z 284.394,A -85,B 0,C 180,E1 -10980.001,E2 -10980.001} C_VEL
LIN {X 0,Y 404.392,Z 284.408,A -85,B 0,C 180,E1 -10982.989,E2 -10982.989} C_VEL
LIN {X 0,Y 404.346,Z 284.42,A -85,B 0,C 180,E1 -10986.545,E2 -10986.545} C_VEL
LIN {X 0,Y 404.266,Z 284.424,A -85,B 0,C 180,E1 -10989.002,E2 -10989.002} C_VEL
LIN {X 0,Y 404.258,Z 284.437,A -85,B 0,C 180,E1 -10992.042,E2 -10992.042} C_VEL
LIN {X 0,Y 404.186,Z 284.442,A -85,B 0,C 180,E1 -10995.119,E2 -10995.119} C_VEL
LIN {X 0,Y 404.169,Z 284.437,A -85,B 0,C 180,E1 -10998.241,E2 -10998.241} C_VEL
LIN {X 0,Y 404.139,Z 284.455,A -85,B 0,C 180,E1 -11001.42,E2 -11001.42} C_VEL
LIN {X 0,Y 404.13,Z 284.446,A -85,B 0,C 180,E1 -11004.669,E2 -11004.669} C_VEL
LIN {X 0,Y 404.101,Z 284.448,A -85,B 0,C 180,E1 -11008.007,E2 -11008.007} C_VEL
LIN {X 0,Y 404.141,Z 284.458,A -85,B 0,C 180,E1 -11010.286,E2 -11010.286} C_VEL
LIN {X 0,Y 404.138,Z 284.46,A -85,B 0,C 180,E1 -11013.814,E2 -11013.814} C_VEL
LIN {X 0,Y 404.132,Z 284.461,A -85,B 0,C 180,E1 -11016.874,E2 -11016.874} C_VEL
LIN {X 0,Y 404.12,Z 284.461,A -85,B 0,C 180,E1 -11020.075,E2 -11020.075} C_VEL
LIN {X 0,Y 404.151,Z 284.628,A -85,B 0,C 180,E1 -11020.66,E2 -11020.66} C_VEL
LIN {X 0,Y 405.637,Z 288.755,A -85,B 0,C 180,E1 -11021.471,E2 -11021.471} C_VEL
LIN {X 0,Y 415.555,Z 305.324,A -85,B 0,C 180,E1 -11022.942,E2 -11022.942} C_VEL
LIN {X 0,Y 424.692,Z 322.681,A -85,B 0,C 180,E1 -11024.248,E2 -11024.248} C_VEL
LIN {X 0,Y 426.753,Z 327.063,A -85,B 0,C 180,E1 -11024.54,E2 -11024.54} C_VEL
LIN {X 0,Y 422.423,Z 494.256,A -85,B 0,C 180,E1 -11027.557,E2 -11027.557} C_VEL
LIN {X 0,Y 421.44,Z 511.276,A -85,B 0,C 180,E1 -11028.06,E2 -11028.06} C_VEL
LIN {X 0,Y 420.304,Z 526.418,A -85,B 0,C 180,E1 -11028.694,E2 -11028.694} C_VEL
LIN {X 0,Y 418.867,Z 541.843,A -85,B 0,C 180,E1 -11029.524,E2 -11029.524} C_VEL
LIN {X 0,Y 417.319,Z 555.77,A -85,B 0,C 180,E1 -11030.451,E2 -11030.451} C_VEL
LIN {X 0,Y 415.38,Z 571.1,A -85,B 0,C 180,E1 -11031.707,E2 -11031.707} C_VEL
LIN {X 0,Y 413.634,Z 584.073,A -85,B 0,C 180,E1 -11032.995,E2 -11032.995} C_VEL
LIN {X 0,Y 411.694,Z 597.126,A -85,B 0,C 180,E1 -11034.52,E2 -11034.52} C_VEL
LIN {X 0,Y 409.872,Z 608.852,A -85,B 0,C 180,E1 -11036.132,E2 -11036.132} C_VEL
LIN {X 0,Y 408.142,Z 620.408,A -85,B 0,C 180,E1 -11038.028,E2 -11038.028} C_VEL
LIN {X 0,Y 406.725,Z 630.107,A -85,B 0,C 180,E1 -11039.927,E2 -11039.927} C_VEL
LIN {X 0,Y 405.525,Z 638.335,A -85,B 0,C 180,E1 -11041.819,E2 -11041.819} C_VEL
LIN {X 0,Y 404.67,Z 645.304,A -85,B 0,C 180,E1 -11043.713,E2 -11043.713} C_VEL
LIN {X 0,Y 403.883,Z 651.792,A -85,B 0,C 180,E1 -11045.862,E2 -11045.862} C_VEL
LIN {X 0,Y 403.379,Z 656.981,A -85,B 0,C 180,E1 -11048.001,E2 -11048.001} C_VEL
LIN {X 0,Y 403.01,Z 661.308,A -85,B 0,C 180,E1 -11050.34,E2 -11050.34} C_VEL
LIN {X 0,Y 402.785,Z 664.323,A -85,B 0,C 180,E1 -11052.745,E2 -11052.745} C_VEL
LIN {X 0,Y 402.771,Z 664.453,A -85,B 0,C 180,E1 -11052.906,E2 -11052.906} C_VEL
LIN {X 0,Y 402.045,Z 665.167,A -85,B 0,C 180,E1 -11053.735,E2 -11053.735} C_VEL
LIN {X 0,Y 399.113,Z 666.017,A -85,B 0,C 180,E1 -11055.085,E2 -11055.085} C_VEL
LIN {X 0,Y 396.699,Z 666.377,A -85,B 0,C 180,E1 -11056.178,E2 -11056.178} C_VEL
LIN {X 0,Y 395.719,Z 666.467,A -85,B 0,C 180,E1 -11057.024,E2 -11057.024} C_VEL
LIN {X 0,Y 395.668,Z 666.405,A -85,B 0,C 180,E1 -11057.311,E2 -11057.311} C_VEL
LIN {X 0,Y 395.641,Z 665.461,A -85,B 0,C 180,E1 -11059.768,E2 -11059.768} C_VEL
LIN {X 0,Y 395.718,Z 663.55,A -85,B 0,C 180,E1 -11061.832,E2 -11061.832} C_VEL
LIN {X 0,Y 395.982,Z 660.658,A -85,B 0,C 180,E1 -11063.887,E2 -11063.887} C_VEL
LIN {X 0,Y 396.179,Z 656.755,A -85,B 0,C 180,E1 -11065.931,E2 -11065.931} C_VEL
LIN {X 0,Y 396.542,Z 651.76,A -85,B 0,C 180,E1 -11067.969,E2 -11067.969} C_VEL
LIN {X 0,Y 397.252,Z 645.663,A -85,B 0,C 180,E1 -11070,E2 -11070} C_VEL
LIN {X 0,Y 398.076,Z 637.245,A -85,B 0,C 180,E1 -11072.276,E2 -11072.276} C_VEL
LIN {X 0,Y 399.323,Z 628.172,A -85,B 0,C 180,E1 -11074.29,E2 -11074.29} C_VEL
LIN {X 0,Y 400.828,Z 617.432,A -85,B 0,C 180,E1 -11076.291,E2 -11076.291} C_VEL
LIN {X 0,Y 402.29,Z 606.395,A -85,B 0,C 180,E1 -11078.034,E2 -11078.034} C_VEL
LIN {X 0,Y 403.883,Z 594.438,A -85,B 0,C 180,E1 -11079.642,E2 -11079.642} C_VEL
LIN {X 0,Y 405.771,Z 580.219,A -85,B 0,C 180,E1 -11081.236,E2 -11081.236} C_VEL
LIN {X 0,Y 407.295,Z 567.187,A -85,B 0,C 180,E1 -11082.456,E2 -11082.456} C_VEL
LIN {X 0,Y 408.866,Z 553.32,A -85,B 0,C 180,E1 -11083.544,E2 -11083.544} C_VEL
LIN {X 0,Y 410.369,Z 537.39,A -85,B 0,C 180,E1 -11084.569,E2 -11084.569} C_VEL
LIN {X 0,Y 411.598,Z 522.005,A -85,B 0,C 180,E1 -11085.347,E2 -11085.347} C_VEL
LIN {X 0,Y 412.658,Z 505.346,A -85,B 0,C 180,E1 -11085.971,E2 -11085.971} C_VEL
LIN {X 0,Y 413.366,Z 489.202,A -85,B 0,C 180,E1 -11086.387,E2 -11086.387} C_VEL
LIN {X 0,Y 417.106,Z 327.56,A -85,B 0,C 180,E1 -11089.256,E2 -11089.256} C_VEL
LIN {X 0,Y 405.104,Z 301.965,A -85,B 0,C 180,E1 -11090.733,E2 -11090.733} C_VEL
LIN {X 0,Y 397.836,Z 287.685,A -85,B 0,C 180,E1 -11091.678,E2 -11091.678} C_VEL
LIN {X 0,Y 397.135,Z 285.317,A -85,B 0,C 180,E1 -11092.124,E2 -11092.124} C_VEL
LIN {X 0,Y 397.097,Z 285.321,A -85,B 0,C 180,E1 -11095.494,E2 -11095.494} C_VEL
LIN {X 0,Y 397.065,Z 285.34,A -85,B 0,C 180,E1 -11098.548,E2 -11098.548} C_VEL
LIN {X 0,Y 397.078,Z 285.334,A -85,B 0,C 180,E1 -11101.834,E2 -11101.834} C_VEL
LIN {X 0,Y 397.117,Z 285.325,A -85,B 0,C 180,E1 -11104.494,E2 -11104.494} C_VEL
LIN {X 0,Y 397.09,Z 285.329,A -85,B 0,C 180,E1 -11108.276,E2 -11108.276} C_VEL
LIN {X 0,Y 397.052,Z 285.332,A -85,B 0,C 180,E1 -11111.976,E2 -11111.976} C_VEL
LIN {X 0,Y 397.086,Z 285.332,A -85,B 0,C 180,E1 -11115.069,E2 -11115.069} C_VEL
LIN {X 0,Y 397.052,Z 285.338,A -85,B 0,C 180,E1 -11118.023,E2 -11118.023} C_VEL
LIN {X 0,Y 397.09,Z 285.309,A -85,B 0,C 180,E1 -11121.723,E2 -11121.723} C_VEL
LIN {X 0,Y 397.118,Z 285.311,A -85,B 0,C 180,E1 -11125.505,E2 -11125.505} C_VEL
LIN {X 0,Y 397.078,Z 285.333,A -85,B 0,C 180,E1 -11129.117,E2 -11129.117} C_VEL
LIN {X 0,Y 397.063,Z 285.336,A -85,B 0,C 180,E1 -11132.251,E2 -11132.251} C_VEL
LIN {X 0,Y 397.105,Z 285.328,A -85,B 0,C 180,E1 -11134.864,E2 -11134.864} C_VEL
LIN {X 0,Y 397.097,Z 285.332,A -85,B 0,C 180,E1 -11138.181,E2 -11138.181} C_VEL
LIN {X 0,Y 397.159,Z 285.317,A -85,B 0,C 180,E1 -11141.426,E2 -11141.426} C_VEL
LIN {X 0,Y 397.179,Z 285.32,A -85,B 0,C 180,E1 -11144.607,E2 -11144.607} C_VEL
LIN {X 0,Y 397.22,Z 285.306,A -85,B 0,C 180,E1 -11147.741,E2 -11147.741} C_VEL
LIN {X 0,Y 397.236,Z 285.314,A -85,B 0,C 180,E1 -11150.837,E2 -11150.837} C_VEL
LIN {X 0,Y 397.366,Z 285.286,A -85,B 0,C 180,E1 -11153.908,E2 -11153.908} C_VEL
LIN {X 0,Y 397.446,Z 285.287,A -85,B 0,C 180,E1 -11157.973,E2 -11157.973} C_VEL
LIN {X 0,Y 397.577,Z 285.257,A -85,B 0,C 180,E1 -11159.999,E2 -11159.999} C_VEL
LIN {X 0,Y 397.375,Z 285.298,A -85,B 0,C 180,E1 -11163.041,E2 -11163.041} C_VEL
LIN {X 0,Y 397.333,Z 285.285,A -85,B 0,C 180,E1 -11167.112,E2 -11167.112} C_VEL
LIN {X 0,Y 397.218,Z 285.316,A -85,B 0,C 180,E1 -11170.19,E2 -11170.19} C_VEL
LIN {X 0,Y 397.226,Z 285.318,A -85,B 0,C 180,E1 -11173.32,E2 -11173.32} C_VEL
LIN {X 0,Y 397.181,Z 285.325,A -85,B 0,C 180,E1 -11177.155,E2 -11177.155} C_VEL
LIN {X 0,Y 397.102,Z 285.334,A -85,B 0,C 180,E1 -11180.729,E2 -11180.729} C_VEL
LIN {X 0,Y 397.132,Z 285.329,A -85,B 0,C 180,E1 -11184.018,E2 -11184.018} C_VEL
LIN {X 0,Y 397.193,Z 285.321,A -85,B 0,C 180,E1 -11187.39,E2 -11187.39} C_VEL
LIN {X 0,Y 397.077,Z 285.336,A -85,B 0,C 180,E1 -11190.882,E2 -11190.882} C_VEL
LIN {X 0,Y 397.124,Z 285.33,A -85,B 0,C 180,E1 -11194.493,E2 -11194.493} C_VEL
LIN {X 0,Y 397.104,Z 285.33,A -85,B 0,C 180,E1 -11198.274,E2 -11198.274} C_VEL
LIN {X 0,Y 397.087,Z 285.327,A -85,B 0,C 180,E1 -11200.908,E2 -11200.908} C_VEL
LIN {X 0,Y 397.102,Z 285.329,A -85,B 0,C 180,E1 -11203.648,E2 -11203.648} C_VEL
LIN {X 0,Y 397.103,Z 285.333,A -85,B 0,C 180,E1 -11206.52,E2 -11206.52} C_VEL
LIN {X 0,Y 397.112,Z 285.333,A -85,B 0,C 180,E1 -11210.423,E2 -11210.423} C_VEL
LIN {X 0,Y 397.123,Z 285.48,A -85,B 0,C 180,E1 -11212.376,E2 -11212.376} C_VEL
LIN {X 0,Y 403.238,Z 304.6,A -85,B 0,C 180,E1 -11215.496,E2 -11215.496} C_VEL
LIN {X 0,Y 404.097,Z 307.469,A -85,B 0,C 180,E1 -11215.915,E2 -11215.915} C_VEL
LIN {X 0,Y 414.179,Z 329.153,A -85,B 0,C 180,E1 -11217.167,E2 -11217.167} C_VEL
LIN {X 0,Y 416.903,Z 345.703,A -85,B 0,C 180,E1 -11217.702,E2 -11217.702} C_VEL
LIN {X 0,Y 413.022,Z 514.679,A -85,B 0,C 180,E1 -11220.711,E2 -11220.711} C_VEL
LIN {X 0,Y 412.087,Z 531.599,A -85,B 0,C 180,E1 -11221.197,E2 -11221.197} C_VEL
LIN {X 0,Y 410.811,Z 548.055,A -85,B 0,C 180,E1 -11221.866,E2 -11221.866} C_VEL
LIN {X 0,Y 409.383,Z 564.113,A -85,B 0,C 180,E1 -11222.732,E2 -11222.732} C_VEL
LIN {X 0,Y 407.846,Z 578.643,A -85,B 0,C 180,E1 -11223.707,E2 -11223.707} C_VEL
LIN {X 0,Y 406.08,Z 593.328,A -85,B 0,C 180,E1 -11224.911,E2 -11224.911} C_VEL
LIN {X 0,Y 404.362,Z 607.284,A -85,B 0,C 180,E1 -11226.302,E2 -11226.302} C_VEL
LIN {X 0,Y 402.645,Z 619.914,A -85,B 0,C 180,E1 -11227.788,E2 -11227.788} C_VEL
LIN {X 0,Y 401.04,Z 632.114,A -85,B 0,C 180,E1 -11229.483,E2 -11229.483} C_VEL
LIN {X 0,Y 399.605,Z 643.102,A -85,B 0,C 180,E1 -11231.279,E2 -11231.279} C_VEL
LIN {X 0,Y 398.364,Z 653.659,A -85,B 0,C 180,E1 -11233.341,E2 -11233.341} C_VEL
LIN {X 0,Y 397.325,Z 662.475,A -85,B 0,C 180,E1 -11235.401,E2 -11235.401} C_VEL
LIN {X 0,Y 396.772,Z 668.705,A -85,B 0,C 180,E1 -11237.11,E2 -11237.11} C_VEL
LIN {X 0,Y 396.22,Z 675.2,A -85,B 0,C 180,E1 -11239.266,E2 -11239.266} C_VEL
LIN {X 0,Y 395.937,Z 680.18,A -85,B 0,C 180,E1 -11241.322,E2 -11241.322} C_VEL
LIN {X 0,Y 395.855,Z 684.79,A -85,B 0,C 180,E1 -11243.833,E2 -11243.833} C_VEL
LIN {X 0,Y 395.741,Z 687.438,A -85,B 0,C 180,E1 -11245.927,E2 -11245.927} C_VEL
LIN {X 0,Y 395.767,Z 688.974,A -85,B 0,C 180,E1 -11247.965,E2 -11247.965} C_VEL
LIN {X 0,Y 395.773,Z 689.568,A -85,B 0,C 180,E1 -11250,E2 -11250} C_VEL
LIN {X 0,Y 395.762,Z 689.154,A -85,B 0,C 180,E1 -11252.035,E2 -11252.035} C_VEL
LIN {X 0,Y 395.737,Z 687.807,A -85,B 0,C 180,E1 -11254.074,E2 -11254.074} C_VEL
LIN {X 0,Y 395.818,Z 685.445,A -85,B 0,C 180,E1 -11256.116,E2 -11256.116} C_VEL
LIN {X 0,Y 395.914,Z 682.112,A -85,B 0,C 180,E1 -11258.164,E2 -11258.164} C_VEL
LIN {X 0,Y 396.117,Z 677.667,A -85,B 0,C 180,E1 -11260.22,E2 -11260.22} C_VEL
LIN {X 0,Y 396.668,Z 672.184,A -85,B 0,C 180,E1 -11262.276,E2 -11262.276} C_VEL
LIN {X 0,Y 397.561,Z 663.538,A -85,B 0,C 180,E1 -11264.852,E2 -11264.852} C_VEL
LIN {X 0,Y 398.765,Z 655.055,A -85,B 0,C 180,E1 -11266.906,E2 -11266.906} C_VEL
LIN {X 0,Y 399.911,Z 646.324,A -85,B 0,C 180,E1 -11268.707,E2 -11268.707} C_VEL
LIN {X 0,Y 401.48,Z 636.238,A -85,B 0,C 180,E1 -11270.494,E2 -11270.494} C_VEL
LIN {X 0,Y 403.326,Z 624.383,A -85,B 0,C 180,E1 -11272.272,E2 -11272.272} C_VEL
LIN {X 0,Y 405.28,Z 611.425,A -85,B 0,C 180,E1 -11273.913,E2 -11273.913} C_VEL
LIN {X 0,Y 407.18,Z 598.565,A -85,B 0,C 180,E1 -11275.29,E2 -11275.29} C_VEL
LIN {X 0,Y 409.185,Z 584.839,A -85,B 0,C 180,E1 -11276.524,E2 -11276.524} C_VEL
LIN {X 0,Y 411.101,Z 569.957,A -85,B 0,C 180,E1 -11277.627,E2 -11277.627} C_VEL
LIN {X 0,Y 412.9,Z 554.677,A -85,B 0,C 180,E1 -11278.532,E2 -11278.532} C_VEL
LIN {X 0,Y 414.367,Z 538.545,A -85,B 0,C 180,E1 -11279.289,E2 -11279.289} C_VEL
LIN {X 0,Y 415.602,Z 523.085,A -85,B 0,C 180,E1 -11279.82,E2 -11279.82} C_VEL
LIN {X 0,Y 416.405,Z 506.47,A -85,B 0,C 180,E1 -11280.21,E2 -11280.21} C_VEL
LIN {X 0,Y 420.63,Z 345.783,A -85,B 0,C 180,E1 -11283.124,E2 -11283.124} C_VEL
LIN {X 0,Y 418.495,Z 332.915,A -85,B 0,C 180,E1 -11283.61,E2 -11283.61} C_VEL
LIN {X 0,Y 411.513,Z 318.837,A -85,B 0,C 180,E1 -11284.649,E2 -11284.649} C_VEL
LIN {X 0,Y 404.785,Z 306.407,A -85,B 0,C 180,E1 -11285.687,E2 -11285.687} C_VEL
LIN {X 0,Y 399.619,Z 292.139,A -85,B 0,C 180,E1 -11288.424,E2 -11288.424} C_VEL
LIN {X 0,Y 397.152,Z 285.322,A -85,B 0,C 180,E1 -11289.822,E2 -11289.822} C_VEL
LIN {X 0,Y 397.103,Z 285.333,A -85,B 0,C 180,E1 -11293.648,E2 -11293.648} C_VEL
LIN {X 0,Y 397.101,Z 285.332,A -85,B 0,C 180,E1 -11296.521,E2 -11296.521} C_VEL
LIN {X 0,Y 397.113,Z 285.331,A -85,B 0,C 180,E1 -11300.423,E2 -11300.423} C_VEL
LIN {X 0,Y 397.108,Z 285.33,A -85,B 0,C 180,E1 -11304.266,E2 -11304.266} C_VEL
LIN {X 0,Y 397.114,Z 285.315,A -85,B 0,C 180,E1 -11306.728,E2 -11306.728} C_VEL
LIN {X 0,Y 397.125,Z 285.326,A -85,B 0,C 180,E1 -11310.296,E2 -11310.296} C_VEL
LIN {X 0,Y 397.195,Z 285.302,A -85,B 0,C 180,E1 -11312.61,E2 -11312.61} C_VEL
LIN {X 0,Y 397.13,Z 285.32,A -85,B 0,C 180,E1 -11315.982,E2 -11315.982} C_VEL
LIN {X 0,Y 397.14,Z 285.326,A -85,B 0,C 180,E1 -11319.705,E2 -11319.705} C_VEL
LIN {X 0,Y 397.183,Z 285.299,A -85,B 0,C 180,E1 -11322.845,E2 -11322.845} C_VEL
LIN {X 0,Y 397.23,Z 285.316,A -85,B 0,C 180,E1 -11326.703,E2 -11326.703} C_VEL
LIN {X 0,Y 397.217,Z 285.293,A -85,B 0,C 180,E1 -11329.81,E2 -11329.81} C_VEL
LIN {X 0,Y 397.297,Z 285.307,A -85,B 0,C 180,E1 -11332.888,E2 -11332.888} C_VEL
LIN {X 0,Y 397.243,Z 285.291,A -85,B 0,C 180,E1 -11334.926,E2 -11334.926} C_VEL
LIN {X 0,Y 397.449,Z 285.285,A -85,B 0,C 180,E1 -11337.974,E2 -11337.974} C_VEL
LIN {X 0,Y 397.574,Z 285.269,A -85,B 0,C 180,E1 -11340.001,E2 -11340.001} C_VEL
LIN {X 0,Y 397.327,Z 285.288,A -85,B 0,C 180,E1 -11343.042,E2 -11343.042} C_VEL
LIN {X 0,Y 397.302,Z 285.297,A -85,B 0,C 180,E1 -11346.538,E2 -11346.538} C_VEL
LIN {X 0,Y 397.237,Z 285.301,A -85,B 0,C 180,E1 -11349.163,E2 -11349.163} C_VEL
LIN {X 0,Y 397.221,Z 285.309,A -85,B 0,C 180,E1 -11352.259,E2 -11352.259} C_VEL
LIN {X 0,Y 397.134,Z 285.322,A -85,B 0,C 180,E1 -11355.394,E2 -11355.394} C_VEL
LIN {X 0,Y 397.117,Z 285.311,A -85,B 0,C 180,E1 -11358.576,E2 -11358.576} C_VEL
LIN {X 0,Y 397.096,Z 285.335,A -85,B 0,C 180,E1 -11361.819,E2 -11361.819} C_VEL
LIN {X 0,Y 397.103,Z 285.327,A -85,B 0,C 180,E1 -11365.136,E2 -11365.136} C_VEL
LIN {X 0,Y 397.062,Z 285.324,A -85,B 0,C 180,E1 -11368.549,E2 -11368.549} C_VEL
LIN {X 0,Y 397.077,Z 285.326,A -85,B 0,C 180,E1 -11371.835,E2 -11371.835} C_VEL
LIN {X 0,Y 397.117,Z 285.33,A -85,B 0,C 180,E1 -11374.495,E2 -11374.495} C_VEL
LIN {X 0,Y 397.09,Z 285.328,A -85,B 0,C 180,E1 -11378.277,E2 -11378.277} C_VEL
LIN {X 0,Y 397.084,Z 285.361,A -85,B 0,C 180,E1 -11379.871,E2 -11379.871} C_VEL
LIN {X 0,Y 398.384,Z 289.019,A -85,B 0,C 180,E1 -11380.61,E2 -11380.61} C_VEL
LIN {X 0,Y 408.985,Z 306.51,A -85,B 0,C 180,E1 -11382.25,E2 -11382.25} C_VEL
LIN {X 0,Y 417.328,Z 321.941,A -85,B 0,C 180,E1 -11383.485,E2 -11383.485} C_VEL
LIN {X 0,Y 420.894,Z 329.171,A -85,B 0,C 180,E1 -11384.004,E2 -11384.004} C_VEL
LIN {X 0,Y 417.306,Z 464.073,A -85,B 0,C 180,E1 -11386.453,E2 -11386.453} C_VEL
LIN {X 0,Y 416.429,Z 495.058,A -85,B 0,C 180,E1 -11387.047,E2 -11387.047} C_VEL
LIN {X 0,Y 415.407,Z 511.895,A -85,B 0,C 180,E1 -11387.555,E2 -11387.555} C_VEL
LIN {X 0,Y 414.238,Z 526.778,A -85,B 0,C 180,E1 -11388.19,E2 -11388.19} C_VEL
LIN {X 0,Y 412.706,Z 542.221,A -85,B 0,C 180,E1 -11389.033,E2 -11389.033} C_VEL
LIN {X 0,Y 410.947,Z 557.393,A -85,B 0,C 180,E1 -11390.07,E2 -11390.07} C_VEL
LIN {X 0,Y 408.971,Z 572.19,A -85,B 0,C 180,E1 -11391.311,E2 -11391.311} C_VEL
LIN {X 0,Y 407.027,Z 585.882,A -85,B 0,C 180,E1 -11392.712,E2 -11392.712} C_VEL
LIN {X 0,Y 405.125,Z 597.795,A -85,B 0,C 180,E1 -11394.143,E2 -11394.143} C_VEL
LIN {X 0,Y 403.203,Z 609.537,A -85,B 0,C 180,E1 -11395.796,E2 -11395.796} C_VEL
LIN {X 0,Y 401.371,Z 621.021,A -85,B 0,C 180,E1 -11397.72,E2 -11397.72} C_VEL
LIN {X 0,Y 399.855,Z 630.76,A -85,B 0,C 180,E1 -11399.67,E2 -11399.67} C_VEL
LIN {X 0,Y 398.622,Z 638.825,A -85,B 0,C 180,E1 -11401.573,E2 -11401.573} C_VEL
LIN {X 0,Y 397.597,Z 646.623,A -85,B 0,C 180,E1 -11403.774,E2 -11403.774} C_VEL
LIN {X 0,Y 396.781,Z 652.936,A -85,B 0,C 180,E1 -11405.959,E2 -11405.959} C_VEL
LIN {X 0,Y 396.287,Z 657.882,A -85,B 0,C 180,E1 -11408.134,E2 -11408.134} C_VEL
LIN {X 0,Y 395.942,Z 661.673,A -85,B 0,C 180,E1 -11410.29,E2 -11410.29} C_VEL
LIN {X 0,Y 395.69,Z 664.316,A -85,B 0,C 180,E1 -11412.425,E2 -11412.425} C_VEL
LIN {X 0,Y 395.616,Z 665.891,A -85,B 0,C 180,E1 -11414.546,E2 -11414.546} C_VEL
LIN {X 0,Y 395.615,Z 666.48,A -85,B 0,C 180,E1 -11416.647,E2 -11416.647} C_VEL
LIN {X 0,Y 395.668,Z 666.405,A -85,B 0,C 180,E1 -11417.311,E2 -11417.311} C_VEL
LIN {X 0,Y 395.061,Z 666.298,A -85,B 0,C 180,E1 -11418.16,E2 -11418.16} C_VEL
LIN {X 0,Y 392.174,Z 665.749,A -85,B 0,C 180,E1 -11419.538,E2 -11419.538} C_VEL
LIN {X 0,Y 389.713,Z 664.997,A -85,B 0,C 180,E1 -11420.648,E2 -11420.648} C_VEL
LIN {X 0,Y 388.69,Z 664.168,A -85,B 0,C 180,E1 -11421.502,E2 -11421.502} C_VEL
LIN {X 0,Y 388.628,Z 663.833,A -85,B 0,C 180,E1 -11421.79,E2 -11421.79} C_VEL
LIN {X 0,Y 388.877,Z 661.193,A -85,B 0,C 180,E1 -11423.775,E2 -11423.775} C_VEL
LIN {X 0,Y 389.218,Z 656.265,A -85,B 0,C 180,E1 -11426.376,E2 -11426.376} C_VEL
LIN {X 0,Y 389.726,Z 649.646,A -85,B 0,C 180,E1 -11428.967,E2 -11428.967} C_VEL
LIN {X 0,Y 390.515,Z 642.964,A -85,B 0,C 180,E1 -11431.031,E2 -11431.031} C_VEL
LIN {X 0,Y 391.411,Z 635.006,A -85,B 0,C 180,E1 -11433.088,E2 -11433.088} C_VEL
LIN {X 0,Y 392.794,Z 625.536,A -85,B 0,C 180,E1 -11435.133,E2 -11435.133} C_VEL
LIN {X 0,Y 394.255,Z 615.785,A -85,B 0,C 180,E1 -11436.911,E2 -11436.911} C_VEL
LIN {X 0,Y 395.822,Z 604.374,A -85,B 0,C 180,E1 -11438.68,E2 -11438.68} C_VEL
LIN {X 0,Y 397.556,Z 591.953,A -85,B 0,C 180,E1 -11440.311,E2 -11440.311} C_VEL
LIN {X 0,Y 399.357,Z 578.458,A -85,B 0,C 180,E1 -11441.805,E2 -11441.805} C_VEL
LIN {X 0,Y 401.019,Z 565.158,A -85,B 0,C 180,E1 -11443.04,E2 -11443.04} C_VEL
LIN {X 0,Y 402.654,Z 550.766,A -85,B 0,C 180,E1 -11444.144,E2 -11444.144} C_VEL
LIN {X 0,Y 404.107,Z 535.182,A -85,B 0,C 180,E1 -11445.122,E2 -11445.122} C_VEL
LIN {X 0,Y 405.381,Z 519.775,A -85,B 0,C 180,E1 -11445.878,E2 -11445.878} C_VEL
LIN {X 0,Y 406.417,Z 503.371,A -85,B 0,C 180,E1 -11446.481,E2 -11446.481} C_VEL
LIN {X 0,Y 407.146,Z 485.9,A -85,B 0,C 180,E1 -11446.903,E2 -11446.903} C_VEL
LIN {X 0,Y 410.825,Z 329.305,A -85,B 0,C 180,E1 -11449.716,E2 -11449.716} C_VEL
LIN {X 0,Y 399.231,Z 304.828,A -85,B 0,C 180,E1 -11451.172,E2 -11451.172} C_VEL
LIN {X 0,Y 390.598,Z 288.076,A -85,B 0,C 180,E1 -11452.297,E2 -11452.297} C_VEL
LIN {X 0,Y 390.072,Z 286.199,A -85,B 0,C 180,E1 -11452.651,E2 -11452.651} C_VEL
LIN {X 0,Y 390.053,Z 286.197,A -85,B 0,C 180,E1 -11455.722,E2 -11455.722} C_VEL
LIN {X 0,Y 390.026,Z 286.214,A -85,B 0,C 180,E1 -11459.112,E2 -11459.112} C_VEL
LIN {X 0,Y 390.041,Z 286.213,A -85,B 0,C 180,E1 -11462.722,E2 -11462.722} C_VEL
LIN {X 0,Y 390.043,Z 286.209,A -85,B 0,C 180,E1 -11465.821,E2 -11465.821} C_VEL
LIN {X 0,Y 390.037,Z 286.208,A -85,B 0,C 180,E1 -11469.211,E2 -11469.211} C_VEL
LIN {X 0,Y 390.031,Z 286.206,A -85,B 0,C 180,E1 -11472.371,E2 -11472.371} C_VEL
LIN {X 0,Y 390.041,Z 286.21,A -85,B 0,C 180,E1 -11475.353,E2 -11475.353} C_VEL
LIN {X 0,Y 390.015,Z 286.217,A -85,B 0,C 180,E1 -11478.184,E2 -11478.184} C_VEL
LIN {X 0,Y 390.058,Z 286.2,A -85,B 0,C 180,E1 -11480.903,E2 -11480.903} C_VEL
LIN {X 0,Y 390.07,Z 286.181,A -85,B 0,C 180,E1 -11484.791,E2 -11484.791} C_VEL
LIN {X 0,Y 390.023,Z 286.212,A -85,B 0,C 180,E1 -11488.495,E2 -11488.495} C_VEL
LIN {X 0,Y 390.016,Z 286.211,A -85,B 0,C 180,E1 -11492.002,E2 -11492.002} C_VEL
LIN {X 0,Y 390.044,Z 286.203,A -85,B 0,C 180,E1 -11495.516,E2 -11495.516} C_VEL
LIN {X 0,Y 390.063,Z 286.207,A -85,B 0,C 180,E1 -11498.878,E2 -11498.878} C_VEL
LIN {X 0,Y 390.113,Z 286.19,A -85,B 0,C 180,E1 -11502.165,E2 -11502.165} C_VEL
LIN {X 0,Y 390.145,Z 286.201,A -85,B 0,C 180,E1 -11505.392,E2 -11505.392} C_VEL
LIN {X 0,Y 390.147,Z 286.185,A -85,B 0,C 180,E1 -11508.571,E2 -11508.571} C_VEL
LIN {X 0,Y 390.271,Z 286.18,A -85,B 0,C 180,E1 -11512.071,E2 -11512.071} C_VEL
LIN {X 0,Y 390.22,Z 286.175,A -85,B 0,C 180,E1 -11514.833,E2 -11514.833} C_VEL
LIN {X 0,Y 390.413,Z 286.163,A -85,B 0,C 180,E1 -11517.936,E2 -11517.936} C_VEL
LIN {X 0,Y 390.547,Z 286.133,A -85,B 0,C 180,E1 -11519.999,E2 -11519.999} C_VEL
LIN {X 0,Y 390.309,Z 286.178,A -85,B 0,C 180,E1 -11523.096,E2 -11523.096} C_VEL
LIN {X 0,Y 390.303,Z 286.163,A -85,B 0,C 180,E1 -11526.202,E2 -11526.202} C_VEL
LIN {X 0,Y 390.277,Z 286.171,A -85,B 0,C 180,E1 -11528.282,E2 -11528.282} C_VEL
LIN {X 0,Y 390.148,Z 286.198,A -85,B 0,C 180,E1 -11531.428,E2 -11531.428} C_VEL
LIN {X 0,Y 390.144,Z 286.199,A -85,B 0,C 180,E1 -11534.607,E2 -11534.607} C_VEL
LIN {X 0,Y 390.111,Z 286.203,A -85,B 0,C 180,E1 -11537.834,E2 -11537.834} C_VEL
LIN {X 0,Y 390.055,Z 286.214,A -85,B 0,C 180,E1 -11541.122,E2 -11541.122} C_VEL
LIN {X 0,Y 390.08,Z 286.208,A -85,B 0,C 180,E1 -11544.48,E2 -11544.48} C_VEL
LIN {X 0,Y 390.116,Z 286.199,A -85,B 0,C 180,E1 -11547.93,E2 -11547.93} C_VEL
LIN {X 0,Y 390.022,Z 286.216,A -85,B 0,C 180,E1 -11551.504,E2 -11551.504} C_VEL
LIN {X 0,Y 390.084,Z 286.204,A -85,B 0,C 180,E1 -11555.206,E2 -11555.206} C_VEL
LIN {X 0,Y 390.09,Z 286.208,A -85,B 0,C 180,E1 -11559.092,E2 -11559.092} C_VEL
LIN {X 0,Y 390.043,Z 286.213,A -85,B 0,C 180,E1 -11562.374,E2 -11562.374} C_VEL
LIN {X 0,Y 390.046,Z 286.212,A -85,B 0,C 180,E1 -11565.355,E2 -11565.355} C_VEL
LIN {X 0,Y 390.031,Z 286.211,A -85,B 0,C 180,E1 -11568.187,E2 -11568.187} C_VEL
LIN {X 0,Y 390.071,Z 286.216,A -85,B 0,C 180,E1 -11571.81,E2 -11571.81} C_VEL
LIN {X 0,Y 396.061,Z 304.9,A -85,B 0,C 180,E1 -11574.939,E2 -11574.939} C_VEL
LIN {X 0,Y 396.849,Z 307.383,A -85,B 0,C 180,E1 -11575.294,E2 -11575.294} C_VEL
LIN {X 0,Y 408.272,Z 331.823,A -85,B 0,C 180,E1 -11576.75,E2 -11576.75} C_VEL
LIN {X 0,Y 410.644,Z 345.876,A -85,B 0,C 180,E1 -11577.219,E2 -11577.219} C_VEL
LIN {X 0,Y 406.741,Z 513.442,A -85,B 0,C 180,E1 -11580.25,E2 -11580.25} C_VEL
LIN {X 0,Y 405.784,Z 529.824,A -85,B 0,C 180,E1 -11580.707,E2 -11580.707} C_VEL
LIN {X 0,Y 404.487,Z 546.737,A -85,B 0,C 180,E1 -11581.386,E2 -11581.386} C_VEL
LIN {X 0,Y 403.1,Z 562.048,A -85,B 0,C 180,E1 -11582.2,E2 -11582.2} C_VEL
LIN {X 0,Y 401.319,Z 578.011,A -85,B 0,C 180,E1 -11583.268,E2 -11583.268} C_VEL
LIN {X 0,Y 399.549,Z 592.53,A -85,B 0,C 180,E1 -11584.472,E2 -11584.472} C_VEL
LIN {X 0,Y 397.985,Z 605.422,A -85,B 0,C 180,E1 -11585.759,E2 -11585.759} C_VEL
LIN {X 0,Y 396.185,Z 617.793,A -85,B 0,C 180,E1 -11587.193,E2 -11587.193} C_VEL
LIN {X 0,Y 394.484,Z 629.903,A -85,B 0,C 180,E1 -11588.853,E2 -11588.853} C_VEL
LIN {X 0,Y 392.921,Z 641.107,A -85,B 0,C 180,E1 -11590.677,E2 -11590.677} C_VEL
LIN {X 0,Y 391.684,Z 650.704,A -85,B 0,C 180,E1 -11592.51,E2 -11592.51} C_VEL
LIN {X 0,Y 390.685,Z 658.975,A -85,B 0,C 180,E1 -11594.346,E2 -11594.346} C_VEL
LIN {X 0,Y 389.81,Z 668.095,A -85,B 0,C 180,E1 -11596.799,E2 -11596.799} C_VEL
LIN {X 0,Y 389.188,Z 674.869,A -85,B 0,C 180,E1 -11599.07,E2 -11599.07} C_VEL
LIN {X 0,Y 388.846,Z 679.882,A -85,B 0,C 180,E1 -11601.163,E2 -11601.163} C_VEL
LIN {X 0,Y 388.798,Z 682.907,A -85,B 0,C 180,E1 -11602.731,E2 -11602.731} C_VEL
LIN {X 0,Y 388.672,Z 686.048,A -85,B 0,C 180,E1 -11604.813,E2 -11604.813} C_VEL
LIN {X 0,Y 388.617,Z 688.076,A -85,B 0,C 180,E1 -11606.89,E2 -11606.89} C_VEL
LIN {X 0,Y 388.698,Z 689.199,A -85,B 0,C 180,E1 -11608.964,E2 -11608.964} C_VEL
LIN {X 0,Y 388.7,Z 689.267,A -85,B 0,C 180,E1 -11611.036,E2 -11611.036} C_VEL
LIN {X 0,Y 388.613,Z 688.446,A -85,B 0,C 180,E1 -11613.11,E2 -11613.11} C_VEL
LIN {X 0,Y 388.658,Z 686.573,A -85,B 0,C 180,E1 -11615.188,E2 -11615.188} C_VEL
LIN {X 0,Y 388.797,Z 683.79,A -85,B 0,C 180,E1 -11617.269,E2 -11617.269} C_VEL
LIN {X 0,Y 388.997,Z 678.814,A -85,B 0,C 180,E1 -11619.883,E2 -11619.883} C_VEL
LIN {X 0,Y 389.671,Z 672.11,A -85,B 0,C 180,E1 -11622.499,E2 -11622.499} C_VEL
LIN {X 0,Y 390.608,Z 663.507,A -85,B 0,C 180,E1 -11625.123,E2 -11625.123} C_VEL
LIN {X 0,Y 392.017,Z 653.926,A -85,B 0,C 180,E1 -11627.475,E2 -11627.475} C_VEL
LIN {X 0,Y 393.496,Z 643.67,A -85,B 0,C 180,E1 -11629.566,E2 -11629.566} C_VEL
LIN {X 0,Y 395.274,Z 633.113,A -85,B 0,C 180,E1 -11631.376,E2 -11631.376} C_VEL
LIN {X 0,Y 397.267,Z 620.971,A -85,B 0,C 180,E1 -11633.152,E2 -11633.152} C_VEL
LIN {X 0,Y 399.321,Z 608.419,A -85,B 0,C 180,E1 -11634.708,E2 -11634.708} C_VEL
LIN {X 0,Y 401.212,Z 596.308,A -85,B 0,C 180,E1 -11635.972,E2 -11635.972} C_VEL
LIN {X 0,Y 403.32,Z 581.704,A -85,B 0,C 180,E1 -11637.261,E2 -11637.261} C_VEL
LIN {X 0,Y 405.357,Z 566.8,A -85,B 0,C 180,E1 -11638.335,E2 -11638.335} C_VEL
LIN {X 0,Y 407.184,Z 550.964,A -85,B 0,C 180,E1 -11639.254,E2 -11639.254} C_VEL
LIN {X 0,Y 408.781,Z 533.677,A -85,B 0,C 180,E1 -11640.013,E2 -11640.013} C_VEL
LIN {X 0,Y 409.967,Z 517.059,A -85,B 0,C 180,E1 -11640.521,E2 -11640.521} C_VEL
LIN {X 0,Y 410.859,Z 492.69,A -85,B 0,C 180,E1 -11641.006,E2 -11641.006} C_VEL
LIN {X 0,Y 414.902,Z 347.377,A -85,B 0,C 180,E1 -11643.672,E2 -11643.672} C_VEL
LIN {X 0,Y 413.186,Z 336.116,A -85,B 0,C 180,E1 -11644.093,E2 -11644.093} C_VEL
LIN {X 0,Y 404.845,Z 319.391,A -85,B 0,C 180,E1 -11645.377,E2 -11645.377} C_VEL
LIN {X 0,Y 397.394,Z 306.02,A -85,B 0,C 180,E1 -11646.582,E2 -11646.582} C_VEL
LIN {X 0,Y 392.467,Z 292.606,A -85,B 0,C 180,E1 -11649.264,E2 -11649.264} C_VEL
LIN {X 0,Y 390.057,Z 286.214,A -85,B 0,C 180,E1 -11650.651,E2 -11650.651} C_VEL
LIN {X 0,Y 390.056,Z 286.21,A -85,B 0,C 180,E1 -11653.887,E2 -11653.887} C_VEL
LIN {X 0,Y 390.056,Z 286.212,A -85,B 0,C 180,E1 -11656.79,E2 -11656.79} C_VEL
LIN {X 0,Y 390.055,Z 286.203,A -85,B 0,C 180,E1 -11659.561,E2 -11659.561} C_VEL
LIN {X 0,Y 390.043,Z 286.197,A -85,B 0,C 180,E1 -11662.45,E2 -11662.45} C_VEL
LIN {X 0,Y 390.068,Z 286.199,A -85,B 0,C 180,E1 -11665.976,E2 -11665.976} C_VEL
LIN {X 0,Y 390.047,Z 286.21,A -85,B 0,C 180,E1 -11669.869,E2 -11669.869} C_VEL
LIN {X 0,Y 390.114,Z 286.192,A -85,B 0,C 180,E1 -11673.232,E2 -11673.232} C_VEL
LIN {X 0,Y 390.077,Z 286.186,A -85,B 0,C 180,E1 -11676.761,E2 -11676.761} C_VEL
LIN {X 0,Y 390.105,Z 286.203,A -85,B 0,C 180,E1 -11679.984,E2 -11679.984} C_VEL
LIN {X 0,Y 390.139,Z 286.175,A -85,B 0,C 180,E1 -11683.249,E2 -11683.249} C_VEL
LIN {X 0,Y 390.196,Z 286.195,A -85,B 0,C 180,E1 -11686.562,E2 -11686.562} C_VEL
LIN {X 0,Y 390.168,Z 286.169,A -85,B 0,C 180,E1 -11689.623,E2 -11689.623} C_VEL
LIN {X 0,Y 390.25,Z 286.187,A -85,B 0,C 180,E1 -11692.758,E2 -11692.758} C_VEL
LIN {X 0,Y 390.213,Z 286.167,A -85,B 0,C 180,E1 -11694.834,E2 -11694.834} C_VEL
LIN {X 0,Y 390.416,Z 286.161,A -85,B 0,C 180,E1 -11697.937,E2 -11697.937} C_VEL
LIN {X 0,Y 390.544,Z 286.144,A -85,B 0,C 180,E1 -11700.001,E2 -11700.001} C_VEL
LIN {X 0,Y 390.263,Z 286.167,A -85,B 0,C 180,E1 -11703.097,E2 -11703.097} C_VEL
LIN {X 0,Y 390.261,Z 286.173,A -85,B 0,C 180,E1 -11706.529,E2 -11706.529} C_VEL
LIN {X 0,Y 390.194,Z 286.18,A -85,B 0,C 180,E1 -11709.33,E2 -11709.33} C_VEL
LIN {X 0,Y 390.173,Z 286.184,A -85,B 0,C 180,E1 -11712.484,E2 -11712.484} C_VEL
LIN {X 0,Y 390.075,Z 286.203,A -85,B 0,C 180,E1 -11715.68,E2 -11715.68} C_VEL
LIN {X 0,Y 390.078,Z 286.186,A -85,B 0,C 180,E1 -11718.924,E2 -11718.924} C_VEL
LIN {X 0,Y 390.037,Z 286.21,A -85,B 0,C 180,E1 -11722.235,E2 -11722.235} C_VEL
LIN {X 0,Y 390.053,Z 286.209,A -85,B 0,C 180,E1 -11725.722,E2 -11725.722} C_VEL
LIN {X 0,Y 390.023,Z 286.206,A -85,B 0,C 180,E1 -11729.113,E2 -11729.113} C_VEL
LIN {X 0,Y 390.041,Z 286.204,A -85,B 0,C 180,E1 -11732.722,E2 -11732.722} C_VEL
LIN {X 0,Y 390.043,Z 286.204,A -85,B 0,C 180,E1 -11735.822,E2 -11735.822} C_VEL
LIN {X 0,Y 390.081,Z 286.339,A -85,B 0,C 180,E1 -11739.094,E2 -11739.094} C_VEL
LIN {X 0,Y 391.196,Z 289.264,A -85,B 0,C 180,E1 -11739.711,E2 -11739.711} C_VEL
LIN {X 0,Y 400.273,Z 304.075,A -85,B 0,C 180,E1 -11741.189,E2 -11741.189} C_VEL
LIN {X 0,Y 408.663,Z 318.774,A -85,B 0,C 180,E1 -11742.486,E2 -11742.486} C_VEL
LIN {X 0,Y 415.194,Z 331.726,A -85,B 0,C 180,E1 -11743.472,E2 -11743.472} C_VEL
LIN {X 0,Y 410.561,Z 493.747,A -85,B 0,C 180,E1 -11746.468,E2 -11746.468} C_VEL
LIN {X 0,Y 409.545,Z 510.135,A -85,B 0,C 180,E1 -11746.948,E2 -11746.948} C_VEL
LIN {X 0,Y 408.335,Z 525.668,A -85,B 0,C 180,E1 -11747.596,E2 -11747.596} C_VEL
LIN {X 0,Y 406.837,Z 540.662,A -85,B 0,C 180,E1 -11748.401,E2 -11748.401} C_VEL
LIN {X 0,Y 405.04,Z 555.567,A -85,B 0,C 180,E1 -11749.408,E2 -11749.408} C_VEL
LIN {X 0,Y 403.017,Z 570.262,A -85,B 0,C 180,E1 -11750.63,E2 -11750.63} C_VEL
LIN {X 0,Y 401.124,Z 582.921,A -85,B 0,C 180,E1 -11751.89,E2 -11751.89} C_VEL
LIN {X 0,Y 399.081,Z 595.622,A -85,B 0,C 180,E1 -11753.376,E2 -11753.376} C_VEL
LIN {X 0,Y 396.917,Z 608.495,A -85,B 0,C 180,E1 -11755.177,E2 -11755.177} C_VEL
LIN {X 0,Y 394.858,Z 620.179,A -85,B 0,C 180,E1 -11757.133,E2 -11757.133} C_VEL
LIN {X 0,Y 393.266,Z 629.878,A -85,B 0,C 180,E1 -11759.072,E2 -11759.072} C_VEL
LIN {X 0,Y 391.885,Z 638.259,A -85,B 0,C 180,E1 -11761.039,E2 -11761.039} C_VEL
LIN {X 0,Y 390.772,Z 646.212,A -85,B 0,C 180,E1 -11763.28,E2 -11763.28} C_VEL
LIN {X 0,Y 389.878,Z 652.603,A -85,B 0,C 180,E1 -11765.506,E2 -11765.506} C_VEL
LIN {X 0,Y 389.281,Z 657.688,A -85,B 0,C 180,E1 -11767.72,E2 -11767.72} C_VEL
LIN {X 0,Y 388.88,Z 661.742,A -85,B 0,C 180,E1 -11770.014,E2 -11770.014} C_VEL
LIN {X 0,Y 388.612,Z 664.315,A -85,B 0,C 180,E1 -11772.095,E2 -11772.095} C_VEL
LIN {X 0,Y 388.525,Z 666.011,A -85,B 0,C 180,E1 -11774.256,E2 -11774.256} C_VEL
LIN {X 0,Y 388.498,Z 666.66,A -85,B 0,C 180,E1 -11776.398,E2 -11776.398} C_VEL
LIN {X 0,Y 388.584,Z 666.318,A -85,B 0,C 180,E1 -11778.524,E2 -11778.524} C_VEL
LIN {X 0,Y 388.55,Z 665.011,A -85,B 0,C 180,E1 -11780.631,E2 -11780.631} C_VEL
LIN {X 0,Y 388.628,Z 663.833,A -85,B 0,C 180,E1 -11781.79,E2 -11781.79} C_VEL
LIN {X 0,Y 388.02,Z 662.851,A -85,B 0,C 180,E1 -11782.643,E2 -11782.643} C_VEL
LIN {X 0,Y 385.24,Z 660.939,A -85,B 0,C 180,E1 -11784.027,E2 -11784.027} C_VEL
LIN {X 0,Y 382.554,Z 658.643,A -85,B 0,C 180,E1 -11785.418,E2 -11785.418} C_VEL
LIN {X 0,Y 382.115,Z 656.951,A -85,B 0,C 180,E1 -11786.272,E2 -11786.272} C_VEL
LIN {X 0,Y 382.501,Z 651.786,A -85,B 0,C 180,E1 -11788.421,E2 -11788.421} C_VEL
LIN {X 0,Y 383.279,Z 645.592,A -85,B 0,C 180,E1 -11790.525,E2 -11790.525} C_VEL
LIN {X 0,Y 384.217,Z 637.099,A -85,B 0,C 180,E1 -11792.883,E2 -11792.883} C_VEL
LIN {X 0,Y 385.629,Z 627.906,A -85,B 0,C 180,E1 -11794.966,E2 -11794.966} C_VEL
LIN {X 0,Y 387.083,Z 618.47,A -85,B 0,C 180,E1 -11796.778,E2 -11796.778} C_VEL
LIN {X 0,Y 388.655,Z 607.544,A -85,B 0,C 180,E1 -11798.58,E2 -11798.58} C_VEL
LIN {X 0,Y 390.249,Z 596.613,A -85,B 0,C 180,E1 -11800.113,E2 -11800.113} C_VEL
LIN {X 0,Y 392.104,Z 583.848,A -85,B 0,C 180,E1 -11801.633,E2 -11801.633} C_VEL
LIN {X 0,Y 393.862,Z 570.103,A -85,B 0,C 180,E1 -11803.019,E2 -11803.019} C_VEL
LIN {X 0,Y 395.544,Z 556.779,A -85,B 0,C 180,E1 -11804.141,E2 -11804.141} C_VEL
LIN {X 0,Y 396.986,Z 542.463,A -85,B 0,C 180,E1 -11805.137,E2 -11805.137} C_VEL
LIN {X 0,Y 398.443,Z 526.948,A -85,B 0,C 180,E1 -11805.998,E2 -11805.998} C_VEL
LIN {X 0,Y 399.594,Z 511.237,A -85,B 0,C 180,E1 -11806.672,E2 -11806.672} C_VEL
LIN {X 0,Y 400.566,Z 494.112,A -85,B 0,C 180,E1 -11807.189,E2 -11807.189} C_VEL
LIN {X 0,Y 404.653,Z 332.108,A -85,B 0,C 180,E1 -11810.158,E2 -11810.158} C_VEL
LIN {X 0,Y 403.894,Z 329.843,A -85,B 0,C 180,E1 -11810.266,E2 -11810.266} C_VEL
LIN {X 0,Y 393.608,Z 308.115,A -85,B 0,C 180,E1 -11811.595,E2 -11811.595} C_VEL
LIN {X 0,Y 384.246,Z 290.246,A -85,B 0,C 180,E1 -11812.832,E2 -11812.832} C_VEL
LIN {X 0,Y 383.267,Z 288.17,A -85,B 0,C 180,E1 -11812.998,E2 -11812.998} C_VEL
LIN {X 0,Y 383.038,Z 287.083,A -85,B 0,C 180,E1 -11813.234,E2 -11813.234} C_VEL
LIN {X 0,Y 382.984,Z 287.077,A -85,B 0,C 180,E1 -11816.13,E2 -11816.13} C_VEL
LIN {X 0,Y 382.977,Z 287.092,A -85,B 0,C 180,E1 -11819.701,E2 -11819.701} C_VEL
LIN {X 0,Y 383.001,Z 287.09,A -85,B 0,C 180,E1 -11823.401,E2 -11823.401} C_VEL
LIN {X 0,Y 383.022,Z 287.087,A -85,B 0,C 180,E1 -11826.161,E2 -11826.161} C_VEL
LIN {X 0,Y 382.986,Z 287.089,A -85,B 0,C 180,E1 -11829.58,E2 -11829.58} C_VEL
LIN {X 0,Y 383.008,Z 287.083,A -85,B 0,C 180,E1 -11832.778,E2 -11832.778} C_VEL
LIN {X 0,Y 382.991,Z 287.083,A -85,B 0,C 180,E1 -11835.787,E2 -11835.787} C_VEL
LIN {X 0,Y 382.963,Z 287.092,A -85,B 0,C 180,E1 -11838.8,E2 -11838.8} C_VEL
LIN {X 0,Y 382.993,Z 287.057,A -85,B 0,C 180,E1 -11842.098,E2 -11842.098} C_VEL
LIN {X 0,Y 383.012,Z 287.065,A -85,B 0,C 180,E1 -11845.331,E2 -11845.331} C_VEL
LIN {X 0,Y 382.982,Z 287.089,A -85,B 0,C 180,E1 -11849.081,E2 -11849.081} C_VEL
LIN {X 0,Y 382.971,Z 287.09,A -85,B 0,C 180,E1 -11852.691,E2 -11852.691} C_VEL
LIN {X 0,Y 383.011,Z 287.074,A -85,B 0,C 180,E1 -11856.191,E2 -11856.191} C_VEL
LIN {X 0,Y 383.062,Z 287.084,A -85,B 0,C 180,E1 -11859.598,E2 -11859.598} C_VEL
LIN {X 0,Y 383.095,Z 287.065,A -85,B 0,C 180,E1 -11862.93,E2 -11862.93} C_VEL
LIN {X 0,Y 383.127,Z 287.068,A -85,B 0,C 180,E1 -11866.463,E2 -11866.463} C_VEL
LIN {X 0,Y 383.144,Z 287.068,A -85,B 0,C 180,E1 -11870.497,E2 -11870.497} C_VEL
LIN {X 0,Y 383.274,Z 287.042,A -85,B 0,C 180,E1 -11873.683,E2 -11873.683} C_VEL
LIN {X 0,Y 383.379,Z 287.04,A -85,B 0,C 180,E1 -11877.898,E2 -11877.898} C_VEL
LIN {X 0,Y 383.516,Z 287.008,A -85,B 0,C 180,E1 -11879.999,E2 -11879.999} C_VEL
LIN {X 0,Y 383.246,Z 287.059,A -85,B 0,C 180,E1 -11883.153,E2 -11883.153} C_VEL
LIN {X 0,Y 383.261,Z 287.04,A -85,B 0,C 180,E1 -11886.316,E2 -11886.316} C_VEL
LIN {X 0,Y 383.222,Z 287.049,A -85,B 0,C 180,E1 -11888.436,E2 -11888.436} C_VEL
LIN {X 0,Y 383.098,Z 287.074,A -85,B 0,C 180,E1 -11891.642,E2 -11891.642} C_VEL
LIN {X 0,Y 383.11,Z 287.077,A -85,B 0,C 180,E1 -11894.881,E2 -11894.881} C_VEL
LIN {X 0,Y 383.052,Z 287.081,A -85,B 0,C 180,E1 -11898.174,E2 -11898.174} C_VEL
LIN {X 0,Y 382.992,Z 287.089,A -85,B 0,C 180,E1 -11901.53,E2 -11901.53} C_VEL
LIN {X 0,Y 383.052,Z 287.084,A -85,B 0,C 180,E1 -11904.96,E2 -11904.96} C_VEL
LIN {X 0,Y 383.016,Z 287.084,A -85,B 0,C 180,E1 -11908.494,E2 -11908.494} C_VEL
LIN {X 0,Y 383.008,Z 287.088,A -85,B 0,C 180,E1 -11912.149,E2 -11912.149} C_VEL
LIN {X 0,Y 383.017,Z 287.089,A -85,B 0,C 180,E1 -11914.667,E2 -11914.667} C_VEL
LIN {X 0,Y 383,Z 287.087,A -85,B 0,C 180,E1 -11917.904,E2 -11917.904} C_VEL
LIN {X 0,Y 382.983,Z 287.086,A -85,B 0,C 180,E1 -11921.347,E2 -11921.347} C_VEL
LIN {X 0,Y 382.997,Z 287.083,A -85,B 0,C 180,E1 -11924.304,E2 -11924.304} C_VEL
LIN {X 0,Y 383.008,Z 287.082,A -85,B 0,C 180,E1 -11927.24,E2 -11927.24} C_VEL
LIN {X 0,Y 383.053,Z 287.189,A -85,B 0,C 180,E1 -11931.26,E2 -11931.26} C_VEL
LIN {X 0,Y 388.348,Z 303.524,A -85,B 0,C 180,E1 -11934.08,E2 -11934.08} C_VEL
LIN {X 0,Y 389.511,Z 307.082,A -85,B 0,C 180,E1 -11934.635,E2 -11934.635} C_VEL
LIN {X 0,Y 402.332,Z 334.416,A -85,B 0,C 180,E1 -11936.317,E2 -11936.317} C_VEL
LIN {X 0,Y 404.479,Z 348.116,A -85,B 0,C 180,E1 -11936.771,E2 -11936.771} C_VEL
LIN {X 0,Y 400.399,Z 513.695,A -85,B 0,C 180,E1 -11939.802,E2 -11939.802} C_VEL
LIN {X 0,Y 399.419,Z 529.907,A -85,B 0,C 180,E1 -11940.266,E2 -11940.266} C_VEL
LIN {X 0,Y 398.196,Z 545.42,A -85,B 0,C 180,E1 -11940.891,E2 -11940.891} C_VEL
LIN {X 0,Y 396.753,Z 560.991,A -85,B 0,C 180,E1 -11941.716,E2 -11941.716} C_VEL
LIN {X 0,Y 395.018,Z 576.201,A -85,B 0,C 180,E1 -11942.734,E2 -11942.734} C_VEL
LIN {X 0,Y 393.233,Z 590.26,A -85,B 0,C 180,E1 -11943.889,E2 -11943.889} C_VEL
LIN {X 0,Y 391.516,Z 603.509,A -85,B 0,C 180,E1 -11945.191,E2 -11945.191} C_VEL
LIN {X 0,Y 389.661,Z 615.951,A -85,B 0,C 180,E1 -11946.622,E2 -11946.622} C_VEL
LIN {X 0,Y 387.739,Z 629.321,A -85,B 0,C 180,E1 -11948.467,E2 -11948.467} C_VEL
LIN {X 0,Y 386.092,Z 640.599,A -85,B 0,C 180,E1 -11950.321,E2 -11950.321} C_VEL
LIN {X 0,Y 384.814,Z 650.26,A -85,B 0,C 180,E1 -11952.187,E2 -11952.187} C_VEL
LIN {X 0,Y 383.607,Z 659.622,A -85,B 0,C 180,E1 -11954.322,E2 -11954.322} C_VEL
LIN {X 0,Y 382.762,Z 668.174,A -85,B 0,C 180,E1 -11956.69,E2 -11956.69} C_VEL
LIN {X 0,Y 382.129,Z 674.526,A -85,B 0,C 180,E1 -11958.866,E2 -11958.866} C_VEL
LIN {X 0,Y 381.776,Z 679.575,A -85,B 0,C 180,E1 -11960.998,E2 -11960.998} C_VEL
LIN {X 0,Y 381.698,Z 682.615,A -85,B 0,C 180,E1 -11962.595,E2 -11962.595} C_VEL
LIN {X 0,Y 381.582,Z 685.786,A -85,B 0,C 180,E1 -11964.716,E2 -11964.716} C_VEL
LIN {X 0,Y 381.528,Z 687.832,A -85,B 0,C 180,E1 -11966.832,E2 -11966.832} C_VEL
LIN {X 0,Y 381.613,Z 688.983,A -85,B 0,C 180,E1 -11968.945,E2 -11968.945} C_VEL
LIN {X 0,Y 381.615,Z 689.066,A -85,B 0,C 180,E1 -11971.055,E2 -11971.055} C_VEL
LIN {X 0,Y 381.524,Z 688.271,A -85,B 0,C 180,E1 -11973.168,E2 -11973.168} C_VEL
LIN {X 0,Y 381.569,Z 686.414,A -85,B 0,C 180,E1 -11975.284,E2 -11975.284} C_VEL
LIN {X 0,Y 381.698,Z 683.66,A -85,B 0,C 180,E1 -11977.405,E2 -11977.405} C_VEL
LIN {X 0,Y 381.942,Z 678.704,A -85,B 0,C 180,E1 -11980.068,E2 -11980.068} C_VEL
LIN {X 0,Y 382.667,Z 672.032,A -85,B 0,C 180,E1 -11982.732,E2 -11982.732} C_VEL
LIN {X 0,Y 383.655,Z 663.486,A -85,B 0,C 180,E1 -11985.404,E2 -11985.404} C_VEL
LIN {X 0,Y 385.144,Z 653.946,A -85,B 0,C 180,E1 -11987.797,E2 -11987.797} C_VEL
LIN {X 0,Y 386.742,Z 643.734,A -85,B 0,C 180,E1 -11989.922,E2 -11989.922} C_VEL
LIN {X 0,Y 388.584,Z 633.233,A -85,B 0,C 180,E1 -11991.763,E2 -11991.763} C_VEL
LIN {X 0,Y 390.697,Z 621.166,A -85,B 0,C 180,E1 -11993.565,E2 -11993.565} C_VEL
LIN {X 0,Y 392.856,Z 608.703,A -85,B 0,C 180,E1 -11995.143,E2 -11995.143} C_VEL
LIN {X 0,Y 394.855,Z 596.675,A -85,B 0,C 180,E1 -11996.422,E2 -11996.422} C_VEL
LIN {X 0,Y 397.143,Z 581.647,A -85,B 0,C 180,E1 -11997.772,E2 -11997.772} C_VEL
LIN {X 0,Y 399.172,Z 567.474,A -85,B 0,C 180,E1 -11998.815,E2 -11998.815} C_VEL
LIN {X 0,Y 401.064,Z 551.796,A -85,B 0,C 180,E1 -11999.744,E2 -11999.744} C_VEL
LIN {X 0,Y 402.65,Z 535.574,A -85,B 0,C 180,E1 -12000.482,E2 -12000.482} C_VEL
LIN {X 0,Y 403.971,Z 518.865,A -85,B 0,C 180,E1 -12001.024,E2 -12001.024} C_VEL
LIN {X 0,Y 404.865,Z 497.366,A -85,B 0,C 180,E1 -12001.481,E2 -12001.481} C_VEL
LIN {X 0,Y 409.211,Z 348.595,A -85,B 0,C 180,E1 -12004.246,E2 -12004.246} C_VEL
LIN {X 0,Y 407.802,Z 339.184,A -85,B 0,C 180,E1 -12004.606,E2 -12004.606} C_VEL
LIN {X 0,Y 401.402,Z 326.21,A -85,B 0,C 180,E1 -12005.619,E2 -12005.619} C_VEL
LIN {X 0,Y 395.089,Z 314.602,A -85,B 0,C 180,E1 -12006.641,E2 -12006.641} C_VEL
LIN {X 0,Y 389.959,Z 305.63,A -85,B 0,C 180,E1 -12007.535,E2 -12007.535} C_VEL
LIN {X 0,Y 385.523,Z 293.608,A -85,B 0,C 180,E1 -12010.036,E2 -12010.036} C_VEL
LIN {X 0,Y 382.99,Z 287.082,A -85,B 0,C 180,E1 -12011.522,E2 -12011.522} C_VEL
LIN {X 0,Y 382.997,Z 287.082,A -85,B 0,C 180,E1 -12014.304,E2 -12014.304} C_VEL
LIN {X 0,Y 383.009,Z 287.086,A -85,B 0,C 180,E1 -12017.241,E2 -12017.241} C_VEL
LIN {X 0,Y 383.015,Z 287.088,A -85,B 0,C 180,E1 -12020.414,E2 -12020.414} C_VEL
LIN {X 0,Y 383.025,Z 287.084,A -85,B 0,C 180,E1 -12024.045,E2 -12024.045} C_VEL
LIN {X 0,Y 382.986,Z 287.075,A -85,B 0,C 180,E1 -12027.579,E2 -12027.579} C_VEL
LIN {X 0,Y 382.992,Z 287.085,A -85,B 0,C 180,E1 -12030.301,E2 -12030.301} C_VEL
LIN {X 0,Y 383.081,Z 287.077,A -85,B 0,C 180,E1 -12034.021,E2 -12034.021} C_VEL
LIN {X 0,Y 382.995,Z 287.065,A -85,B 0,C 180,E1 -12037.335,E2 -12037.335} C_VEL
LIN {X 0,Y 383.061,Z 287.081,A -85,B 0,C 180,E1 -12040.717,E2 -12040.717} C_VEL
LIN {X 0,Y 383.081,Z 287.058,A -85,B 0,C 180,E1 -12044.027,E2 -12044.027} C_VEL
LIN {X 0,Y 383.137,Z 287.066,A -85,B 0,C 180,E1 -12047.285,E2 -12047.285} C_VEL
LIN {X 0,Y 383.144,Z 287.051,A -85,B 0,C 180,E1 -12050.498,E2 -12050.498} C_VEL
LIN {X 0,Y 383.244,Z 287.055,A -85,B 0,C 180,E1 -12053.684,E2 -12053.684} C_VEL
LIN {X 0,Y 383.382,Z 287.036,A -85,B 0,C 180,E1 -12057.899,E2 -12057.899} C_VEL
LIN {X 0,Y 383.514,Z 287.019,A -85,B 0,C 180,E1 -12060.001,E2 -12060.001} C_VEL
LIN {X 0,Y 383.376,Z 287.015,A -85,B 0,C 180,E1 -12062.102,E2 -12062.102} C_VEL
LIN {X 0,Y 383.226,Z 287.049,A -85,B 0,C 180,E1 -12066.517,E2 -12066.517} C_VEL
LIN {X 0,Y 383.144,Z 287.061,A -85,B 0,C 180,E1 -12069.503,E2 -12069.503} C_VEL
LIN {X 0,Y 383.139,Z 287.057,A -85,B 0,C 180,E1 -12072.717,E2 -12072.717} C_VEL
LIN {X 0,Y 383.027,Z 287.083,A -85,B 0,C 180,E1 -12075.976,E2 -12075.976} C_VEL
LIN {X 0,Y 383.045,Z 287.061,A -85,B 0,C 180,E1 -12079.285,E2 -12079.285} C_VEL
LIN {X 0,Y 382.987,Z 287.084,A -85,B 0,C 180,E1 -12082.667,E2 -12082.667} C_VEL
LIN {X 0,Y 382.984,Z 287.095,A -85,B 0,C 180,E1 -12086.131,E2 -12086.131} C_VEL
LIN {X 0,Y 382.975,Z 287.09,A -85,B 0,C 180,E1 -12089.702,E2 -12089.702} C_VEL
LIN {X 0,Y 383.001,Z 287.09,A -85,B 0,C 180,E1 -12093.402,E2 -12093.402} C_VEL
LIN {X 0,Y 383.023,Z 287.081,A -85,B 0,C 180,E1 -12096.162,E2 -12096.162} C_VEL
LIN {X 0,Y 383.024,Z 287.27,A -85,B 0,C 180,E1 -12098.253,E2 -12098.253} C_VEL
LIN {X 0,Y 383.749,Z 289.43,A -85,B 0,C 180,E1 -12098.723,E2 -12098.723} C_VEL
LIN {X 0,Y 390.349,Z 299.768,A -85,B 0,C 180,E1 -12099.856,E2 -12099.856} C_VEL
LIN {X 0,Y 398.746,Z 313.636,A -85,B 0,C 180,E1 -12101.227,E2 -12101.227} C_VEL
LIN {X 0,Y 406.619,Z 328.159,A -85,B 0,C 180,E1 -12102.467,E2 -12102.467} C_VEL
LIN {X 0,Y 409.547,Z 334.375,A -85,B 0,C 180,E1 -12102.927,E2 -12102.927} C_VEL
LIN {X 0,Y 404.668,Z 494.452,A -85,B 0,C 180,E1 -12105.919,E2 -12105.919} C_VEL
LIN {X 0,Y 403.602,Z 510.855,A -85,B 0,C 180,E1 -12106.413,E2 -12106.413} C_VEL
LIN {X 0,Y 402.342,Z 526.083,A -85,B 0,C 180,E1 -12107.059,E2 -12107.059} C_VEL
LIN {X 0,Y 400.682,Z 541.798,A -85,B 0,C 180,E1 -12107.922,E2 -12107.922} C_VEL
LIN {X 0,Y 398.791,Z 556.93,A -85,B 0,C 180,E1 -12108.969,E2 -12108.969} C_VEL
LIN {X 0,Y 396.651,Z 571.59,A -85,B 0,C 180,E1 -12110.221,E2 -12110.221} C_VEL
LIN {X 0,Y 394.501,Z 585.107,A -85,B 0,C 180,E1 -12111.616,E2 -12111.616} C_VEL
LIN {X 0,Y 392.386,Z 597.494,A -85,B 0,C 180,E1 -12113.129,E2 -12113.129} C_VEL
LIN {X 0,Y 390.301,Z 609.235,A -85,B 0,C 180,E1 -12114.815,E2 -12114.815} C_VEL
LIN {X 0,Y 388.093,Z 621.123,A -85,B 0,C 180,E1 -12116.852,E2 -12116.852} C_VEL
LIN {X 0,Y 386.256,Z 631.667,A -85,B 0,C 180,E1 -12119.035,E2 -12119.035} C_VEL
LIN {X 0,Y 384.709,Z 640.627,A -85,B 0,C 180,E1 -12121.27,E2 -12121.27} C_VEL
LIN {X 0,Y 383.692,Z 647.505,A -85,B 0,C 180,E1 -12123.336,E2 -12123.336} C_VEL
LIN {X 0,Y 382.768,Z 653.745,A -85,B 0,C 180,E1 -12125.599,E2 -12125.599} C_VEL
LIN {X 0,Y 382.206,Z 658.598,A -85,B 0,C 180,E1 -12127.855,E2 -12127.855} C_VEL
LIN {X 0,Y 381.816,Z 661.967,A -85,B 0,C 180,E1 -12129.844,E2 -12129.844} C_VEL
LIN {X 0,Y 381.57,Z 664.316,A -85,B 0,C 180,E1 -12131.753,E2 -12131.753} C_VEL
LIN {X 0,Y 381.452,Z 666.133,A -85,B 0,C 180,E1 -12133.956,E2 -12133.956} C_VEL
LIN {X 0,Y 381.385,Z 666.841,A -85,B 0,C 180,E1 -12136.139,E2 -12136.139} C_VEL
LIN {X 0,Y 381.504,Z 666.614,A -85,B 0,C 180,E1 -12138.308,E2 -12138.308} C_VEL
LIN {X 0,Y 381.448,Z 665.364,A -85,B 0,C 180,E1 -12140.455,E2 -12140.455} C_VEL
LIN {X 0,Y 381.638,Z 663.164,A -85,B 0,C 180,E1 -12142.593,E2 -12142.593} C_VEL
LIN {X 0,Y 381.882,Z 659.939,A -85,B 0,C 180,E1 -12144.72,E2 -12144.72} C_VEL
LIN {X 0,Y 382.115,Z 656.951,A -85,B 0,C 180,E1 -12146.272,E2 -12146.272} C_VEL
LIN {X 0,Y 381.701,Z 655.21,A -85,B 0,C 180,E1 -12147.114,E2 -12147.114} C_VEL
LIN {X 0,Y 379.183,Z 652.125,A -85,B 0,C 180,E1 -12148.48,E2 -12148.48} C_VEL
LIN {X 0,Y 377.039,Z 649.317,A -85,B 0,C 180,E1 -12149.564,E2 -12149.564} C_VEL
LIN {X 0,Y 376.246,Z 646.903,A -85,B 0,C 180,E1 -12150.381,E2 -12150.381} C_VEL
LIN {X 0,Y 376.256,Z 646.031,A -85,B 0,C 180,E1 -12150.651,E2 -12150.651} C_VEL
LIN {X 0,Y 377.323,Z 636.98,A -85,B 0,C 180,E1 -12153.203,E2 -12153.203} C_VEL
LIN {X 0,Y 378.782,Z 627.754,A -85,B 0,C 180,E1 -12155.323,E2 -12155.323} C_VEL
LIN {X 0,Y 380.327,Z 618.241,A -85,B 0,C 180,E1 -12157.165,E2 -12157.165} C_VEL
LIN {X 0,Y 381.978,Z 607.23,A -85,B 0,C 180,E1 -12158.997,E2 -12158.997} C_VEL
LIN {X 0,Y 383.832,Z 595.277,A -85,B 0,C 180,E1 -12160.684,E2 -12160.684} C_VEL
LIN {X 0,Y 385.727,Z 582.216,A -85,B 0,C 180,E1 -12162.228,E2 -12162.228} C_VEL
LIN {X 0,Y 387.441,Z 569.44,A -85,B 0,C 180,E1 -12163.506,E2 -12163.506} C_VEL
LIN {X 0,Y 389.379,Z 554.212,A -85,B 0,C 180,E1 -12164.77,E2 -12164.77} C_VEL
LIN {X 0,Y 390.943,Z 539.433,A -85,B 0,C 180,E1 -12165.777,E2 -12165.777} C_VEL
LIN {X 0,Y 392.298,Z 524.252,A -85,B 0,C 180,E1 -12166.59,E2 -12166.59} C_VEL
LIN {X 0,Y 393.439,Z 508.258,A -85,B 0,C 180,E1 -12167.242,E2 -12167.242} C_VEL
LIN {X 0,Y 394.381,Z 490.586,A -85,B 0,C 180,E1 -12167.735,E2 -12167.735} C_VEL
LIN {X 0,Y 398.478,Z 334.147,A -85,B 0,C 180,E1 -12170.63,E2 -12170.63} C_VEL
LIN {X 0,Y 397.234,Z 330.83,A -85,B 0,C 180,E1 -12170.804,E2 -12170.804} C_VEL
LIN {X 0,Y 387.252,Z 309.942,A -85,B 0,C 180,E1 -12172.126,E2 -12172.126} C_VEL
LIN {X 0,Y 378.893,Z 294.011,A -85,B 0,C 180,E1 -12173.263,E2 -12173.263} C_VEL
LIN {X 0,Y 377.303,Z 291.302,A -85,B 0,C 180,E1 -12173.48,E2 -12173.48} C_VEL
LIN {X 0,Y 376.056,Z 288.427,A -85,B 0,C 180,E1 -12173.686,E2 -12173.686} C_VEL
LIN {X 0,Y 375.98,Z 287.971,A -85,B 0,C 180,E1 -12173.817,E2 -12173.817} C_VEL
LIN {X 0,Y 375.913,Z 287.961,A -85,B 0,C 180,E1 -12176.66,E2 -12176.66} C_VEL
LIN {X 0,Y 375.916,Z 287.972,A -85,B 0,C 180,E1 -12179.084,E2 -12179.084} C_VEL
LIN {X 0,Y 375.938,Z 287.969,A -85,B 0,C 180,E1 -12181.564,E2 -12181.564} C_VEL
LIN {X 0,Y 375.977,Z 287.957,A -85,B 0,C 180,E1 -12184.665,E2 -12184.665} C_VEL
LIN {X 0,Y 375.935,Z 287.963,A -85,B 0,C 180,E1 -12188.262,E2 -12188.262} C_VEL
LIN {X 0,Y 375.915,Z 287.965,A -85,B 0,C 180,E1 -12191.596,E2 -12191.596} C_VEL
LIN {X 0,Y 375.921,Z 287.969,A -85,B 0,C 180,E1 -12194.73,E2 -12194.73} C_VEL
LIN {X 0,Y 375.909,Z 287.966,A -85,B 0,C 180,E1 -12197.696,E2 -12197.696} C_VEL
LIN {X 0,Y 375.935,Z 287.96,A -85,B 0,C 180,E1 -12200.533,E2 -12200.533} C_VEL
LIN {X 0,Y 375.958,Z 287.922,A -85,B 0,C 180,E1 -12203.497,E2 -12203.497} C_VEL
LIN {X 0,Y 375.959,Z 287.949,A -85,B 0,C 180,E1 -12205.888,E2 -12205.888} C_VEL
LIN {X 0,Y 375.962,Z 287.959,A -85,B 0,C 180,E1 -12209.686,E2 -12209.686} C_VEL
LIN {X 0,Y 375.919,Z 287.968,A -85,B 0,C 180,E1 -12212.134,E2 -12212.134} C_VEL
LIN {X 0,Y 375.969,Z 287.954,A -85,B 0,C 180,E1 -12215.716,E2 -12215.716} C_VEL
LIN {X 0,Y 376,Z 287.961,A -85,B 0,C 180,E1 -12219.197,E2 -12219.197} C_VEL
LIN {X 0,Y 376.034,Z 287.944,A -85,B 0,C 180,E1 -12222.6,E2 -12222.6} C_VEL
LIN {X 0,Y 376.091,Z 287.945,A -85,B 0,C 180,E1 -12226.342,E2 -12226.342} C_VEL
LIN {X 0,Y 376.114,Z 287.945,A -85,B 0,C 180,E1 -12230.318,E2 -12230.318} C_VEL
LIN {X 0,Y 376.23,Z 287.92,A -85,B 0,C 180,E1 -12233.564,E2 -12233.564} C_VEL
LIN {X 0,Y 376.344,Z 287.917,A -85,B 0,C 180,E1 -12237.859,E2 -12237.859} C_VEL
LIN {X 0,Y 376.486,Z 287.884,A -85,B 0,C 180,E1 -12239.999,E2 -12239.999} C_VEL
LIN {X 0,Y 376.184,Z 287.939,A -85,B 0,C 180,E1 -12243.212,E2 -12243.212} C_VEL
LIN {X 0,Y 376.221,Z 287.915,A -85,B 0,C 180,E1 -12246.435,E2 -12246.435} C_VEL
LIN {X 0,Y 376.119,Z 287.947,A -85,B 0,C 180,E1 -12249.681,E2 -12249.681} C_VEL
LIN {X 0,Y 376.089,Z 287.951,A -85,B 0,C 180,E1 -12253.657,E2 -12253.657} C_VEL
LIN {X 0,Y 376.032,Z 287.961,A -85,B 0,C 180,E1 -12257.399,E2 -12257.399} C_VEL
LIN {X 0,Y 375.977,Z 287.967,A -85,B 0,C 180,E1 -12260.832,E2 -12260.832} C_VEL
LIN {X 0,Y 375.993,Z 287.963,A -85,B 0,C 180,E1 -12264.281,E2 -12264.281} C_VEL
LIN {X 0,Y 376.019,Z 287.961,A -85,B 0,C 180,E1 -12266.652,E2 -12266.652} C_VEL
LIN {X 0,Y 375.963,Z 287.966,A -85,B 0,C 180,E1 -12270.312,E2 -12270.312} C_VEL
LIN {X 0,Y 375.958,Z 287.965,A -85,B 0,C 180,E1 -12274.111,E2 -12274.111} C_VEL
LIN {X 0,Y 375.953,Z 287.955,A -85,B 0,C 180,E1 -12276.741,E2 -12276.741} C_VEL
LIN {X 0,Y 375.987,Z 287.96,A -85,B 0,C 180,E1 -12279.97,E2 -12279.97} C_VEL
LIN {X 0,Y 375.93,Z 287.966,A -85,B 0,C 180,E1 -12283.765,E2 -12283.765} C_VEL
LIN {X 0,Y 375.933,Z 287.966,A -85,B 0,C 180,E1 -12286.81,E2 -12286.81} C_VEL
LIN {X 0,Y 375.994,Z 287.991,A -85,B 0,C 180,E1 -12290.658,E2 -12290.658} C_VEL
LIN {X 0,Y 382.132,Z 306.817,A -85,B 0,C 180,E1 -12293.947,E2 -12293.947} C_VEL
LIN {X 0,Y 394.255,Z 332.261,A -85,B 0,C 180,E1 -12295.589,E2 -12295.589} C_VEL
LIN {X 0,Y 396.539,Z 337.519,A -85,B 0,C 180,E1 -12295.894,E2 -12295.894} C_VEL
LIN {X 0,Y 398.305,Z 348.619,A -85,B 0,C 180,E1 -12296.273,E2 -12296.273} C_VEL
LIN {X 0,Y 394.077,Z 513.705,A -85,B 0,C 180,E1 -12299.34,E2 -12299.34} C_VEL
LIN {X 0,Y 393.072,Z 529.842,A -85,B 0,C 180,E1 -12299.81,E2 -12299.81} C_VEL
LIN {X 0,Y 391.8,Z 545.326,A -85,B 0,C 180,E1 -12300.443,E2 -12300.443} C_VEL
LIN {X 0,Y 390.311,Z 560.887,A -85,B 0,C 180,E1 -12301.279,E2 -12301.279} C_VEL
LIN {X 0,Y 388.429,Z 576.795,A -85,B 0,C 180,E1 -12302.362,E2 -12302.362} C_VEL
LIN {X 0,Y 386.555,Z 590.878,A -85,B 0,C 180,E1 -12303.549,E2 -12303.549} C_VEL
LIN {X 0,Y 384.783,Z 603.99,A -85,B 0,C 180,E1 -12304.871,E2 -12304.871} C_VEL
LIN {X 0,Y 382.77,Z 616.933,A -85,B 0,C 180,E1 -12306.404,E2 -12306.404} C_VEL
LIN {X 0,Y 381.036,Z 628.731,A -85,B 0,C 180,E1 -12308.068,E2 -12308.068} C_VEL
LIN {X 0,Y 379.279,Z 640.072,A -85,B 0,C 180,E1 -12309.952,E2 -12309.952} C_VEL
LIN {X 0,Y 377.958,Z 649.789,A -85,B 0,C 180,E1 -12311.853,E2 -12311.853} C_VEL
LIN {X 0,Y 376.64,Z 659.203,A -85,B 0,C 180,E1 -12314.024,E2 -12314.024} C_VEL
LIN {X 0,Y 375.778,Z 667.564,A -85,B 0,C 180,E1 -12316.367,E2 -12316.367} C_VEL
LIN {X 0,Y 375.08,Z 674.182,A -85,B 0,C 180,E1 -12318.654,E2 -12318.654} C_VEL
LIN {X 0,Y 374.716,Z 679.267,A -85,B 0,C 180,E1 -12320.827,E2 -12320.827} C_VEL
LIN {X 0,Y 374.615,Z 682.324,A -85,B 0,C 180,E1 -12322.454,E2 -12322.454} C_VEL
LIN {X 0,Y 374.498,Z 685.518,A -85,B 0,C 180,E1 -12324.616,E2 -12324.616} C_VEL
LIN {X 0,Y 374.442,Z 687.588,A -85,B 0,C 180,E1 -12326.772,E2 -12326.772} C_VEL
LIN {X 0,Y 374.514,Z 688.762,A -85,B 0,C 180,E1 -12328.925,E2 -12328.925} C_VEL
LIN {X 0,Y 374.515,Z 688.865,A -85,B 0,C 180,E1 -12331.075,E2 -12331.075} C_VEL
LIN {X 0,Y 374.438,Z 688.091,A -85,B 0,C 180,E1 -12333.228,E2 -12333.228} C_VEL
LIN {X 0,Y 374.552,Z 685.573,A -85,B 0,C 180,E1 -12336.028,E2 -12336.028} C_VEL
LIN {X 0,Y 374.615,Z 683.527,A -85,B 0,C 180,E1 -12337.546,E2 -12337.546} C_VEL
LIN {X 0,Y 374.876,Z 678.598,A -85,B 0,C 180,E1 -12340.259,E2 -12340.259} C_VEL
LIN {X 0,Y 375.455,Z 673.399,A -85,B 0,C 180,E1 -12342.431,E2 -12342.431} C_VEL
LIN {X 0,Y 376.181,Z 667.096,A -85,B 0,C 180,E1 -12344.609,E2 -12344.609} C_VEL
LIN {X 0,Y 377.565,Z 658.428,A -85,B 0,C 180,E1 -12347.048,E2 -12347.048} C_VEL
LIN {X 0,Y 379.31,Z 647.855,A -85,B 0,C 180,E1 -12349.482,E2 -12349.482} C_VEL
LIN {X 0,Y 381.413,Z 636.567,A -85,B 0,C 180,E1 -12351.625,E2 -12351.625} C_VEL
LIN {X 0,Y 383.501,Z 625.019,A -85,B 0,C 180,E1 -12353.467,E2 -12353.467} C_VEL
LIN {X 0,Y 385.836,Z 612.164,A -85,B 0,C 180,E1 -12355.2,E2 -12355.2} C_VEL
LIN {X 0,Y 388.036,Z 599.607,A -85,B 0,C 180,E1 -12356.633,E2 -12356.633} C_VEL
LIN {X 0,Y 390.262,Z 586.152,A -85,B 0,C 180,E1 -12357.919,E2 -12357.919} C_VEL
LIN {X 0,Y 392.452,Z 571.667,A -85,B 0,C 180,E1 -12359.062,E2 -12359.062} C_VEL
LIN {X 0,Y 394.604,Z 555.966,A -85,B 0,C 180,E1 -12360.061,E2 -12360.061} C_VEL
LIN {X 0,Y 396.249,Z 540.558,A -85,B 0,C 180,E1 -12360.843,E2 -12360.843} C_VEL
LIN {X 0,Y 397.799,Z 524.065,A -85,B 0,C 180,E1 -12361.449,E2 -12361.449} C_VEL
LIN {X 0,Y 398.754,Z 506.68,A -85,B 0,C 180,E1 -12361.884,E2 -12361.884} C_VEL
LIN {X 0,Y 403.531,Z 349.055,A -85,B 0,C 180,E1 -12364.86,E2 -12364.86} C_VEL
LIN {X 0,Y 402.424,Z 342.127,A -85,B 0,C 180,E1 -12365.14,E2 -12365.14} C_VEL
LIN {X 0,Y 393.642,Z 324.512,A -85,B 0,C 180,E1 -12366.585,E2 -12366.585} C_VEL
LIN {X 0,Y 384.947,Z 309.501,A -85,B 0,C 180,E1 -12368.062,E2 -12368.062} C_VEL
LIN {X 0,Y 382.601,Z 305.345,A -85,B 0,C 180,E1 -12368.517,E2 -12368.517} C_VEL
LIN {X 0,Y 378.109,Z 293.65,A -85,B 0,C 180,E1 -12371.08,E2 -12371.08} C_VEL
LIN {X 0,Y 375.956,Z 287.957,A -85,B 0,C 180,E1 -12372.427,E2 -12372.427} C_VEL
LIN {X 0,Y 375.93,Z 287.966,A -85,B 0,C 180,E1 -12376.235,E2 -12376.235} C_VEL
LIN {X 0,Y 375.988,Z 287.962,A -85,B 0,C 180,E1 -12380.03,E2 -12380.03} C_VEL
LIN {X 0,Y 375.963,Z 287.955,A -85,B 0,C 180,E1 -12383.496,E2 -12383.496} C_VEL
LIN {X 0,Y 375.959,Z 287.956,A -85,B 0,C 180,E1 -12385.889,E2 -12385.889} C_VEL
LIN {X 0,Y 375.965,Z 287.964,A -85,B 0,C 180,E1 -12389.688,E2 -12389.688} C_VEL
LIN {X 0,Y 376.02,Z 287.948,A -85,B 0,C 180,E1 -12393.349,E2 -12393.349} C_VEL
LIN {X 0,Y 375.984,Z 287.939,A -85,B 0,C 180,E1 -12396.888,E2 -12396.888} C_VEL
LIN {X 0,Y 375.999,Z 287.963,A -85,B 0,C 180,E1 -12400.34,E2 -12400.34} C_VEL
LIN {X 0,Y 376.029,Z 287.932,A -85,B 0,C 180,E1 -12403.719,E2 -12403.719} C_VEL
LIN {X 0,Y 376.105,Z 287.944,A -85,B 0,C 180,E1 -12407.043,E2 -12407.043} C_VEL
LIN {X 0,Y 376.114,Z 287.924,A -85,B 0,C 180,E1 -12410.319,E2 -12410.319} C_VEL
LIN {X 0,Y 376.202,Z 287.932,A -85,B 0,C 180,E1 -12413.565,E2 -12413.565} C_VEL
LIN {X 0,Y 376.347,Z 287.913,A -85,B 0,C 180,E1 -12417.86,E2 -12417.86} C_VEL
LIN {X 0,Y 376.462,Z 287.897,A -85,B 0,C 180,E1 -12420.001,E2 -12420.001} C_VEL
LIN {X 0,Y 376.34,Z 287.891,A -85,B 0,C 180,E1 -12422.141,E2 -12422.141} C_VEL
LIN {X 0,Y 376.195,Z 287.925,A -85,B 0,C 180,E1 -12426.502,E2 -12426.502} C_VEL
LIN {X 0,Y 376.115,Z 287.938,A -85,B 0,C 180,E1 -12429.682,E2 -12429.682} C_VEL
LIN {X 0,Y 376.092,Z 287.926,A -85,B 0,C 180,E1 -12433.658,E2 -12433.658} C_VEL
LIN {X 0,Y 376.01,Z 287.954,A -85,B 0,C 180,E1 -12437.59,E2 -12437.59} C_VEL
LIN {X 0,Y 375.982,Z 287.96,A -85,B 0,C 180,E1 -12440.833,E2 -12440.833} C_VEL
LIN {X 0,Y 375.934,Z 287.952,A -85,B 0,C 180,E1 -12444.286,E2 -12444.286} C_VEL
LIN {X 0,Y 375.912,Z 287.97,A -85,B 0,C 180,E1 -12446.661,E2 -12446.661} C_VEL
LIN {X 0,Y 375.914,Z 287.961,A -85,B 0,C 180,E1 -12449.085,E2 -12449.085} C_VEL
LIN {X 0,Y 375.937,Z 287.959,A -85,B 0,C 180,E1 -12451.565,E2 -12451.565} C_VEL
LIN {X 0,Y 375.977,Z 287.96,A -85,B 0,C 180,E1 -12454.666,E2 -12454.666} C_VEL
LIN {X 0,Y 375.96,Z 288.013,A -85,B 0,C 180,E1 -12457.328,E2 -12457.328} C_VEL
LIN {X 0,Y 376.424,Z 289.754,A -85,B 0,C 180,E1 -12457.696,E2 -12457.696} C_VEL
LIN {X 0,Y 383.887,Z 301.1,A -85,B 0,C 180,E1 -12459.034,E2 -12459.034} C_VEL
LIN {X 0,Y 391.666,Z 313.85,A -85,B 0,C 180,E1 -12460.363,E2 -12460.363} C_VEL
LIN {X 0,Y 399.95,Z 328.69,A -85,B 0,C 180,E1 -12461.717,E2 -12461.717} C_VEL
LIN {X 0,Y 403.827,Z 336.413,A -85,B 0,C 180,E1 -12462.339,E2 -12462.339} C_VEL
LIN {X 0,Y 398.858,Z 494.626,A -85,B 0,C 180,E1 -12465.341,E2 -12465.341} C_VEL
LIN {X 0,Y 397.774,Z 510.755,A -85,B 0,C 180,E1 -12465.829,E2 -12465.829} C_VEL
LIN {X 0,Y 396.39,Z 526.845,A -85,B 0,C 180,E1 -12466.522,E2 -12466.522} C_VEL
LIN {X 0,Y 394.628,Z 542.643,A -85,B 0,C 180,E1 -12467.41,E2 -12467.41} C_VEL
LIN {X 0,Y 392.809,Z 556.476,A -85,B 0,C 180,E1 -12468.377,E2 -12468.377} C_VEL
LIN {X 0,Y 390.595,Z 571.054,A -85,B 0,C 180,E1 -12469.628,E2 -12469.628} C_VEL
LIN {X 0,Y 388.371,Z 584.514,A -85,B 0,C 180,E1 -12471.019,E2 -12471.019} C_VEL
LIN {X 0,Y 386.051,Z 597.303,A -85,B 0,C 180,E1 -12472.585,E2 -12472.585} C_VEL
LIN {X 0,Y 384.037,Z 608.157,A -85,B 0,C 180,E1 -12474.154,E2 -12474.154} C_VEL
LIN {X 0,Y 381.93,Z 619.084,A -85,B 0,C 180,E1 -12476.012,E2 -12476.012} C_VEL
LIN {X 0,Y 380.03,Z 629.2,A -85,B 0,C 180,E1 -12478.048,E2 -12478.048} C_VEL
LIN {X 0,Y 378.361,Z 638.232,A -85,B 0,C 180,E1 -12480.207,E2 -12480.207} C_VEL
LIN {X 0,Y 376.877,Z 647.116,A -85,B 0,C 180,E1 -12482.814,E2 -12482.814} C_VEL
LIN {X 0,Y 375.883,Z 653.442,A -85,B 0,C 180,E1 -12485.122,E2 -12485.122} C_VEL
LIN {X 0,Y 375.211,Z 658.417,A -85,B 0,C 180,E1 -12487.419,E2 -12487.419} C_VEL
LIN {X 0,Y 374.782,Z 662.18,A -85,B 0,C 180,E1 -12489.656,E2 -12489.656} C_VEL
LIN {X 0,Y 374.421,Z 665.409,A -85,B 0,C 180,E1 -12492.523,E2 -12492.523} C_VEL
LIN {X 0,Y 374.311,Z 666.735,A -85,B 0,C 180,E1 -12494.76,E2 -12494.76} C_VEL
LIN {X 0,Y 374.437,Z 667.006,A -85,B 0,C 180,E1 -12497.429,E2 -12497.429} C_VEL
LIN {X 0,Y 374.387,Z 666.421,A -85,B 0,C 180,E1 -12499.18,E2 -12499.18} C_VEL
LIN {X 0,Y 374.407,Z 664.789,A -85,B 0,C 180,E1 -12501.363,E2 -12501.363} C_VEL
LIN {X 0,Y 374.709,Z 661.875,A -85,B 0,C 180,E1 -12503.759,E2 -12503.759} C_VEL
LIN {X 0,Y 375.036,Z 657.291,A -85,B 0,C 180,E1 -12506.32,E2 -12506.32} C_VEL
LIN {X 0,Y 375.41,Z 652.494,A -85,B 0,C 180,E1 -12508.391,E2 -12508.391} C_VEL
LIN {X 0,Y 376.256,Z 646.031,A -85,B 0,C 180,E1 -12510.651,E2 -12510.651} C_VEL
LIN {X 0,Y 375.889,Z 643.46,A -85,B 0,C 180,E1 -12511.457,E2 -12511.457} C_VEL
LIN {X 0,Y 371.484,Z 634.535,A -85,B 0,C 180,E1 -12514.09,E2 -12514.09} C_VEL
LIN {X 0,Y 371.387,Z 631.353,A -85,B 0,C 180,E1 -12514.856,E2 -12514.856} C_VEL
LIN {X 0,Y 373.147,Z 620.916,A -85,B 0,C 180,E1 -12517.032,E2 -12517.032} C_VEL
LIN {X 0,Y 374.797,Z 610.273,A -85,B 0,C 180,E1 -12518.899,E2 -12518.899} C_VEL
LIN {X 0,Y 376.806,Z 597.748,A -85,B 0,C 180,E1 -12520.749,E2 -12520.749} C_VEL
LIN {X 0,Y 378.753,Z 585.123,A -85,B 0,C 180,E1 -12522.321,E2 -12522.321} C_VEL
LIN {X 0,Y 380.653,Z 571.54,A -85,B 0,C 180,E1 -12523.751,E2 -12523.751} C_VEL
LIN {X 0,Y 382.649,Z 556.747,A -85,B 0,C 180,E1 -12525.036,E2 -12525.036} C_VEL
LIN {X 0,Y 384.458,Z 540.362,A -85,B 0,C 180,E1 -12526.187,E2 -12526.187} C_VEL
LIN {X 0,Y 385.885,Z 525.349,A -85,B 0,C 180,E1 -12527.01,E2 -12527.01} C_VEL
LIN {X 0,Y 387.105,Z 508.838,A -85,B 0,C 180,E1 -12527.704,E2 -12527.704} C_VEL
LIN {X 0,Y 388.025,Z 492.86,A -85,B 0,C 180,E1 -12528.172,E2 -12528.172} C_VEL
LIN {X 0,Y 392.3,Z 336.354,A -85,B 0,C 180,E1 -12531.114,E2 -12531.114} C_VEL
LIN {X 0,Y 391.629,Z 334.165,A -85,B 0,C 180,E1 -12531.219,E2 -12531.219} C_VEL
LIN {X 0,Y 382.048,Z 313.952,A -85,B 0,C 180,E1 -12532.521,E2 -12532.521} C_VEL
LIN {X 0,Y 373.021,Z 296.604,A -85,B 0,C 180,E1 -12533.785,E2 -12533.785} C_VEL
LIN {X 0,Y 369.217,Z 290.162,A -85,B 0,C 180,E1 -12534.319,E2 -12534.319} C_VEL
LIN {X 0,Y 368.915,Z 288.845,A -85,B 0,C 180,E1 -12534.382,E2 -12534.382} C_VEL
LIN {X 0,Y 368.86,Z 288.847,A -85,B 0,C 180,E1 -12537.212,E2 -12537.212} C_VEL
LIN {X 0,Y 368.895,Z 288.846,A -85,B 0,C 180,E1 -12539.692,E2 -12539.692} C_VEL
LIN {X 0,Y 368.897,Z 288.848,A -85,B 0,C 180,E1 -12543.538,E2 -12543.538} C_VEL
LIN {X 0,Y 368.897,Z 288.845,A -85,B 0,C 180,E1 -12546.854,E2 -12546.854} C_VEL
LIN {X 0,Y 368.886,Z 288.847,A -85,B 0,C 180,E1 -12550.373,E2 -12550.373} C_VEL
LIN {X 0,Y 368.88,Z 288.846,A -85,B 0,C 180,E1 -12553.614,E2 -12553.614} C_VEL
LIN {X 0,Y 368.884,Z 288.836,A -85,B 0,C 180,E1 -12556.695,E2 -12556.695} C_VEL
LIN {X 0,Y 368.886,Z 288.847,A -85,B 0,C 180,E1 -12559.648,E2 -12559.648} C_VEL
LIN {X 0,Y 368.896,Z 288.8,A -85,B 0,C 180,E1 -12563.145,E2 -12563.145} C_VEL
LIN {X 0,Y 368.897,Z 288.839,A -85,B 0,C 180,E1 -12566.461,E2 -12566.461} C_VEL
LIN {X 0,Y 368.914,Z 288.842,A -85,B 0,C 180,E1 -12569.044,E2 -12569.044} C_VEL
LIN {X 0,Y 368.908,Z 288.833,A -85,B 0,C 180,E1 -12571.557,E2 -12571.557} C_VEL
LIN {X 0,Y 368.924,Z 288.837,A -85,B 0,C 180,E1 -12575.222,E2 -12575.222} C_VEL
LIN {X 0,Y 368.921,Z 288.841,A -85,B 0,C 180,E1 -12578.98,E2 -12578.98} C_VEL
LIN {X 0,Y 368.992,Z 288.82,A -85,B 0,C 180,E1 -12582.257,E2 -12582.257} C_VEL
LIN {X 0,Y 369.039,Z 288.824,A -85,B 0,C 180,E1 -12586.227,E2 -12586.227} C_VEL
LIN {X 0,Y 369.064,Z 288.824,A -85,B 0,C 180,E1 -12590.131,E2 -12590.131} C_VEL
LIN {X 0,Y 369.189,Z 288.797,A -85,B 0,C 180,E1 -12593.441,E2 -12593.441} C_VEL
LIN {X 0,Y 369.308,Z 288.793,A -85,B 0,C 180,E1 -12597.818,E2 -12597.818} C_VEL
LIN {X 0,Y 369.455,Z 288.759,A -85,B 0,C 180,E1 -12599.999,E2 -12599.999} C_VEL
LIN {X 0,Y 369.317,Z 288.79,A -85,B 0,C 180,E1 -12602.181,E2 -12602.181} C_VEL
LIN {X 0,Y 369.183,Z 288.79,A -85,B 0,C 180,E1 -12606.558,E2 -12606.558} C_VEL
LIN {X 0,Y 369.107,Z 288.808,A -85,B 0,C 180,E1 -12608.761,E2 -12608.761} C_VEL
LIN {X 0,Y 369.005,Z 288.827,A -85,B 0,C 180,E1 -12612.093,E2 -12612.093} C_VEL
LIN {X 0,Y 368.996,Z 288.831,A -85,B 0,C 180,E1 -12615.464,E2 -12615.464} C_VEL
LIN {X 0,Y 368.953,Z 288.839,A -85,B 0,C 180,E1 -12618.894,E2 -12618.894} C_VEL
LIN {X 0,Y 368.931,Z 288.838,A -85,B 0,C 180,E1 -12622.395,E2 -12622.395} C_VEL
LIN {X 0,Y 368.999,Z 288.833,A -85,B 0,C 180,E1 -12625.98,E2 -12625.98} C_VEL
LIN {X 0,Y 368.913,Z 288.844,A -85,B 0,C 180,E1 -12629.69,E2 -12629.69} C_VEL
LIN {X 0,Y 368.895,Z 288.846,A -85,B 0,C 180,E1 -12633.043,E2 -12633.043} C_VEL
LIN {X 0,Y 368.916,Z 288.833,A -85,B 0,C 180,E1 -12636.196,E2 -12636.196} C_VEL
LIN {X 0,Y 368.903,Z 288.849,A -85,B 0,C 180,E1 -12638.952,E2 -12638.952} C_VEL
LIN {X 0,Y 368.88,Z 288.848,A -85,B 0,C 180,E1 -12642.009,E2 -12642.009} C_VEL
LIN {X 0,Y 368.926,Z 288.839,A -85,B 0,C 180,E1 -12645.183,E2 -12645.183} C_VEL
LIN {X 0,Y 368.882,Z 288.845,A -85,B 0,C 180,E1 -12648.178,E2 -12648.178} C_VEL
LIN {X 0,Y 368.965,Z 288.924,A -85,B 0,C 180,E1 -12650.056,E2 -12650.056} C_VEL
LIN {X 0,Y 374.78,Z 306.614,A -85,B 0,C 180,E1 -12653.234,E2 -12653.234} C_VEL
LIN {X 0,Y 384.489,Z 326.618,A -85,B 0,C 180,E1 -12654.598,E2 -12654.598} C_VEL
LIN {X 0,Y 390.692,Z 340.495,A -85,B 0,C 180,E1 -12655.451,E2 -12655.451} C_VEL
LIN {X 0,Y 392.138,Z 350.287,A -85,B 0,C 180,E1 -12655.784,E2 -12655.784} C_VEL
LIN {X 0,Y 387.774,Z 513.898,A -85,B 0,C 180,E1 -12658.867,E2 -12658.867} C_VEL
LIN {X 0,Y 386.656,Z 530.692,A -85,B 0,C 180,E1 -12659.369,E2 -12659.369} C_VEL
LIN {X 0,Y 385.314,Z 546.533,A -85,B 0,C 180,E1 -12660.046,E2 -12660.046} C_VEL
LIN {X 0,Y 383.638,Z 562.765,A -85,B 0,C 180,E1 -12660.957,E2 -12660.957} C_VEL
LIN {X 0,Y 381.738,Z 578.117,A -85,B 0,C 180,E1 -12662.043,E2 -12662.043} C_VEL
LIN {X 0,Y 379.67,Z 592.891,A -85,B 0,C 180,E1 -12663.328,E2 -12663.328} C_VEL
LIN {X 0,Y 377.764,Z 606.823,A -85,B 0,C 180,E1 -12664.813,E2 -12664.813} C_VEL
LIN {X 0,Y 375.823,Z 618.403,A -85,B 0,C 180,E1 -12666.253,E2 -12666.253} C_VEL
LIN {X 0,Y 374.043,Z 629.921,A -85,B 0,C 180,E1 -12667.927,E2 -12667.927} C_VEL
LIN {X 0,Y 372.256,Z 641.057,A -85,B 0,C 180,E1 -12669.846,E2 -12669.846} C_VEL
LIN {X 0,Y 370.891,Z 650.57,A -85,B 0,C 180,E1 -12671.781,E2 -12671.781} C_VEL
LIN {X 0,Y 369.569,Z 659.807,A -85,B 0,C 180,E1 -12673.994,E2 -12673.994} C_VEL
LIN {X 0,Y 368.751,Z 667.431,A -85,B 0,C 180,E1 -12676.183,E2 -12676.183} C_VEL
LIN {X 0,Y 368.041,Z 673.823,A -85,B 0,C 180,E1 -12678.434,E2 -12678.434} C_VEL
LIN {X 0,Y 367.637,Z 678.948,A -85,B 0,C 180,E1 -12680.649,E2 -12680.649} C_VEL
LIN {X 0,Y 367.475,Z 683.767,A -85,B 0,C 180,E1 -12683.411,E2 -12683.411} C_VEL
LIN {X 0,Y 367.418,Z 686.407,A -85,B 0,C 180,E1 -12685.612,E2 -12685.612} C_VEL
LIN {X 0,Y 367.363,Z 688.057,A -85,B 0,C 180,E1 -12687.807,E2 -12687.807} C_VEL
LIN {X 0,Y 367.452,Z 688.71,A -85,B 0,C 180,E1 -12690,E2 -12690} C_VEL
LIN {X 0,Y 367.355,Z 688.406,A -85,B 0,C 180,E1 -12692.193,E2 -12692.193} C_VEL
LIN {X 0,Y 367.393,Z 687.116,A -85,B 0,C 180,E1 -12694.389,E2 -12694.389} C_VEL
LIN {X 0,Y 367.474,Z 684.873,A -85,B 0,C 180,E1 -12696.589,E2 -12696.589} C_VEL
LIN {X 0,Y 367.599,Z 681.605,A -85,B 0,C 180,E1 -12698.798,E2 -12698.798} C_VEL
LIN {X 0,Y 367.97,Z 677.299,A -85,B 0,C 180,E1 -12701.011,E2 -12701.011} C_VEL
LIN {X 0,Y 368.647,Z 671.9,A -85,B 0,C 180,E1 -12703.225,E2 -12703.225} C_VEL
LIN {X 0,Y 369.518,Z 665.258,A -85,B 0,C 180,E1 -12705.443,E2 -12705.443} C_VEL
LIN {X 0,Y 371.106,Z 656.231,A -85,B 0,C 180,E1 -12707.923,E2 -12707.923} C_VEL
LIN {X 0,Y 372.755,Z 646.604,A -85,B 0,C 180,E1 -12710.126,E2 -12710.126} C_VEL
LIN {X 0,Y 375.03,Z 635.157,A -85,B 0,C 180,E1 -12712.302,E2 -12712.302} C_VEL
LIN {X 0,Y 377.32,Z 623.297,A -85,B 0,C 180,E1 -12714.191,E2 -12714.191} C_VEL
LIN {X 0,Y 379.604,Z 611.378,A -85,B 0,C 180,E1 -12715.791,E2 -12715.791} C_VEL
LIN {X 0,Y 381.724,Z 600,A -85,B 0,C 180,E1 -12717.109,E2 -12717.109} C_VEL
LIN {X 0,Y 384.284,Z 585.152,A -85,B 0,C 180,E1 -12718.548,E2 -12718.548} C_VEL
LIN {X 0,Y 386.604,Z 570.566,A -85,B 0,C 180,E1 -12719.695,E2 -12719.695} C_VEL
LIN {X 0,Y 388.763,Z 554.63,A -85,B 0,C 180,E1 -12720.711,E2 -12720.711} C_VEL
LIN {X 0,Y 390.606,Z 538.069,A -85,B 0,C 180,E1 -12721.528,E2 -12721.528} C_VEL
LIN {X 0,Y 392.092,Z 521.708,A -85,B 0,C 180,E1 -12722.112,E2 -12722.112} C_VEL
LIN {X 0,Y 393.027,Z 505.243,A -85,B 0,C 180,E1 -12722.511,E2 -12722.511} C_VEL
LIN {X 0,Y 397.978,Z 350.444,A -85,B 0,C 180,E1 -12725.463,E2 -12725.463} C_VEL
LIN {X 0,Y 396.989,Z 344.82,A -85,B 0,C 180,E1 -12725.708,E2 -12725.708} C_VEL
LIN {X 0,Y 388.622,Z 328.171,A -85,B 0,C 180,E1 -12727.127,E2 -12727.127} C_VEL
LIN {X 0,Y 380.386,Z 313.796,A -85,B 0,C 180,E1 -12728.573,E2 -12728.573} C_VEL
LIN {X 0,Y 375.221,Z 305.081,A -85,B 0,C 180,E1 -12729.556,E2 -12729.556} C_VEL
LIN {X 0,Y 370.935,Z 294.22,A -85,B 0,C 180,E1 -12732.06,E2 -12732.06} C_VEL
LIN {X 0,Y 368.892,Z 288.848,A -85,B 0,C 180,E1 -12733.38,E2 -12733.38} C_VEL
LIN {X 0,Y 368.885,Z 288.848,A -85,B 0,C 180,E1 -12736.697,E2 -12736.697} C_VEL
LIN {X 0,Y 368.911,Z 288.836,A -85,B 0,C 180,E1 -12739.644,E2 -12739.644} C_VEL
LIN {X 0,Y 368.901,Z 288.831,A -85,B 0,C 180,E1 -12743.145,E2 -12743.145} C_VEL
LIN {X 0,Y 368.896,Z 288.829,A -85,B 0,C 180,E1 -12746.463,E2 -12746.463} C_VEL
LIN {X 0,Y 368.929,Z 288.842,A -85,B 0,C 180,E1 -12749.047,E2 -12749.047} C_VEL
LIN {X 0,Y 368.963,Z 288.818,A -85,B 0,C 180,E1 -12752.797,E2 -12752.797} C_VEL
LIN {X 0,Y 368.937,Z 288.825,A -85,B 0,C 180,E1 -12756.116,E2 -12756.116} C_VEL
LIN {X 0,Y 368.938,Z 288.84,A -85,B 0,C 180,E1 -12759.948,E2 -12759.948} C_VEL
LIN {X 0,Y 368.976,Z 288.809,A -85,B 0,C 180,E1 -12763.399,E2 -12763.399} C_VEL
LIN {X 0,Y 369.059,Z 288.824,A -85,B 0,C 180,E1 -12766.791,E2 -12766.791} C_VEL
LIN {X 0,Y 369.064,Z 288.799,A -85,B 0,C 180,E1 -12770.132,E2 -12770.132} C_VEL
LIN {X 0,Y 369.163,Z 288.809,A -85,B 0,C 180,E1 -12773.442,E2 -12773.442} C_VEL
LIN {X 0,Y 369.311,Z 288.789,A -85,B 0,C 180,E1 -12777.819,E2 -12777.819} C_VEL
LIN {X 0,Y 369.413,Z 288.774,A -85,B 0,C 180,E1 -12780.001,E2 -12780.001} C_VEL
LIN {X 0,Y 369.304,Z 288.767,A -85,B 0,C 180,E1 -12782.182,E2 -12782.182} C_VEL
LIN {X 0,Y 369.163,Z 288.8,A -85,B 0,C 180,E1 -12786.56,E2 -12786.56} C_VEL
LIN {X 0,Y 369.065,Z 288.817,A -85,B 0,C 180,E1 -12789.869,E2 -12789.869} C_VEL
LIN {X 0,Y 369.04,Z 288.804,A -85,B 0,C 180,E1 -12793.773,E2 -12793.773} C_VEL
LIN {X 0,Y 368.956,Z 288.828,A -85,B 0,C 180,E1 -12797.745,E2 -12797.745} C_VEL
LIN {X 0,Y 368.912,Z 288.844,A -85,B 0,C 180,E1 -12801.221,E2 -12801.221} C_VEL
LIN {X 0,Y 368.907,Z 288.826,A -85,B 0,C 180,E1 -12803.873,E2 -12803.873} C_VEL
LIN {X 0,Y 368.858,Z 288.842,A -85,B 0,C 180,E1 -12807.213,E2 -12807.213} C_VEL
LIN {X 0,Y 368.894,Z 288.844,A -85,B 0,C 180,E1 -12809.693,E2 -12809.693} C_VEL
LIN {X 0,Y 368.897,Z 288.848,A -85,B 0,C 180,E1 -12813.539,E2 -12813.539} C_VEL
LIN {X 0,Y 368.942,Z 289.009,A -85,B 0,C 180,E1 -12816.407,E2 -12816.407} C_VEL
LIN {X 0,Y 369.214,Z 290.162,A -85,B 0,C 180,E1 -12816.623,E2 -12816.623} C_VEL
LIN {X 0,Y 370.643,Z 292.663,A -85,B 0,C 180,E1 -12816.91,E2 -12816.91} C_VEL
LIN {X 0,Y 372.27,Z 294.608,A -85,B 0,C 180,E1 -12817.209,E2 -12817.209} C_VEL
LIN {X 0,Y 380.113,Z 306.659,A -85,B 0,C 180,E1 -12818.656,E2 -12818.656} C_VEL
LIN {X 0,Y 388.478,Z 320.472,A -85,B 0,C 180,E1 -12820.117,E2 -12820.117} C_VEL
LIN {X 0,Y 396.841,Z 336.069,A -85,B 0,C 180,E1 -12821.52,E2 -12821.52} C_VEL
LIN {X 0,Y 398.25,Z 338.976,A -85,B 0,C 180,E1 -12821.754,E2 -12821.754} C_VEL
LIN {X 0,Y 393.083,Z 495.129,A -85,B 0,C 180,E1 -12824.754,E2 -12824.754} C_VEL
LIN {X 0,Y 391.917,Z 511.634,A -85,B 0,C 180,E1 -12825.263,E2 -12825.263} C_VEL
LIN {X 0,Y 390.474,Z 527.567,A -85,B 0,C 180,E1 -12825.966,E2 -12825.966} C_VEL
LIN {X 0,Y 388.494,Z 544.26,A -85,B 0,C 180,E1 -12826.928,E2 -12826.928} C_VEL
LIN {X 0,Y 386.363,Z 559.435,A -85,B 0,C 180,E1 -12828.038,E2 -12828.038} C_VEL
LIN {X 0,Y 384.066,Z 573.749,A -85,B 0,C 180,E1 -12829.315,E2 -12829.315} C_VEL
LIN {X 0,Y 381.574,Z 588.021,A -85,B 0,C 180,E1 -12830.871,E2 -12830.871} C_VEL
LIN {X 0,Y 379.404,Z 599.2,A -85,B 0,C 180,E1 -12832.317,E2 -12832.317} C_VEL
LIN {X 0,Y 377.104,Z 610.717,A -85,B 0,C 180,E1 -12834.051,E2 -12834.051} C_VEL
LIN {X 0,Y 374.774,Z 622.126,A -85,B 0,C 180,E1 -12836.09,E2 -12836.09} C_VEL
LIN {X 0,Y 372.882,Z 631.708,A -85,B 0,C 180,E1 -12838.147,E2 -12838.147} C_VEL
LIN {X 0,Y 371.31,Z 639.823,A -85,B 0,C 180,E1 -12840.208,E2 -12840.208} C_VEL
